# B&R Automation Studio project NAEUL004C00R13L518F00 (part 13)

#### Act_OptP0202InsertRmvMag.st
```iecst
ACTION Act_OptP0202InsertRmvMag:

	//Insert & Removed Magazine Manually Without Button Control
//	IF p_tyNtParamCurr.bProjBtnInsertRmvMag = FALSE THEN
//
//		IF p_bOpsStatusRun AND p_bOpsMagConvUL1InitDone THEN
//
//			fbMag1EntrySenOnTm(IN := p_tyDI.bMagPresentSen1 OR p_tyDI.bMagConvEntSen1);
//
//			IF bNewMag1 = FALSE AND bRlsMag1 = FALSE THEN
//				IF p_bOpsMagConvUL1NewMagAllw AND fbMag1EntrySenOnTm.Q AND NOT p_bOpsMagConvUL1MagExitedWait THEN
//					bNewMag1	:= TRUE;
//				END_IF
//
//				IF p_bOpsMagConvUL1RlsMagAllw AND p_tyDI.bMagPresentSen1 AND p_tyDI.bOutShutterCloseRS AND p_tyBuffer1BffrStat.bBffrFull THEN
//					bRlsMag1	:= TRUE;
//				END_IF
//			END_IF
//
//			IF bNewMag1 = TRUE THEN
//
//				IF p_tyDI.bMag1FixedClampRS = TRUE AND p_tyDI.bMag1RemoteClampRS = TRUE THEN
//					bNewMag1	:= FALSE;
//				END_IF
//
//			ELSIF bRlsMag1 = TRUE THEN
//
//				IF p_tyDI.bMag1FixedUnclampRS = TRUE AND p_tyDI.bMag1RemoteUnclampRS = TRUE AND p_tyDI.bMagConvEntSen1 = TRUE THEN
//					bRlsMag1	:= FALSE;
//				END_IF
//
//			END_IF
//
//		ELSE
//
//			bNewMag1	:= FALSE;
//			bRlsMag1	:= FALSE;
//
//			fbMag1EntrySenOnTm(IN := FALSE);
//
//		END_IF
//
//	END_IF

END_ACTION
```

#### Act_OptP0202RstMnl.st
```iecst
ACTION Act_OptP0202RstMnl:

	IF eCurrPage <> UIP0202OpsMag1 AND eCurrPage <> UIP0003MMenu THEN
		bNewMag1	:= FALSE;
		bRlsMag1	:= FALSE;
		tyP0202OpsMag1.tyOps.tyBtnChgMag.bValue	:= FALSE;
		tyP0202OpsMag1.tyOps.tyBtnChgMag.bRtLk	:= FALSE;
		tyP0202OpsMag1.tyOps.tyBitmapChgMag.usiValueIdx	:= 0;

		tyP0003MMenu.tyMMenuBtn.tyBtnRlsNewMag1.bValue := FALSE;
		tyP0003MMenu.tyMMenuBtn.tyBtnRlsNewMag1.bRtLk  := FALSE;
		tyP0003MMenu.tyMMenuBtn.tyBtnRlsNewMag1.usiBitmapIdx := 0;
	END_IF

END_ACTION
```

#### Act_OptP0202Lane1ChgMag.st
```iecst
ACTION Act_OptP0202Lane1ChgMag:

	tyP0202OpsMag1.tyChgMag.tyBtnChgMag.bRtLk				:= FALSE;

	tChgMag ( IN:= tyP0202OpsMag1.tyChgMag.tyBtnChgMag.bValue = TRUE OR  FALSE , PT:=T#3s0ms);

	IF tChgMag.IN = TRUE THEN

	fbChgMagBlinkTm(IN := TRUE);

		IF fbChgMagBlinkTm.Q THEN
			fbChgMagBlinkTm(IN := FALSE);

			IF (tyP0202OpsMag1.tyChgMag.tyBitmapChgMag.usiValueIdx = 1) THEN
				tyP0202OpsMag1.tyChgMag.tyBitmapChgMag.usiValueIdx		:= 0;
			ELSE
				tyP0202OpsMag1.tyChgMag.tyBitmapChgMag.usiValueIdx		:= 1;
			END_IF
		END_IF
	ELSIF bChgMag = FALSE THEN

		tyP0202OpsMag1.tyChgMag.tyBitmapChgMag.usiValueIdx		:= 0;
	END_IF

	IF tChgMag.Q = TRUE THEN //(tyP0200OpsGen.tyChgMag.tyBtnChgMag.bRtCompl = TRUE) OR (tyP0202OpsMag1.tyChgMag.tyBtnChgMag.bRtCompl = TRUE)
	//	OR (tyP0203OpsMag2.tyChgMag.tyBtnChgMag.bRtCompl = TRUE)	OR (tyP0204OpsOutMagConv.tyChgMag.tyBtnChgMag.bRtCompl = TRUE) THEN

		tyP0202OpsMag1.tyChgMag.tyBitmapChgMag.usiValueIdx	:= 1;

		tyP0202OpsMag1.tyChgMag.tyBtnChgMag.bRtCompl			:= FALSE;

		bChgMag			:= TRUE;

//	ELSIF EDGEPOS(p_bFollower2SetBffrFull) THEN
//		bFllw2SetFull	:= TRUE;
//	ELSIF EDGEPOS(p_tyDI.bChgMagSig) THEN
//		bChgMagSig		:= TRUE;
	END_IF

	IF (p_bOpsOutMagConvStepInitDone AND p_bOpsStatusRun = TRUE) AND bChgMag = TRUE THEN

		eBuffer1Act			:= BufferActSetFull;

		IF p_eBuffer1Stat = BufferActSetFull AND p_eBuffer1Status = Done THEN
			eBuffer1Act		:= BufferActIdle;

			bChgMag			:= FALSE;

		END_IF

//	ELSIF bFllw2SetFull = TRUE THEN
//		eBufferAct			:= BufferActSetFull;
//
//		IF p_eBufferStat = BufferActSetFull AND p_eBufferStatus = Done THEN
//			eBufferAct		:= BufferActIdle;
//
//			bFllw2SetFull	:= FALSE;
//		END_IF

	ELSIF (p_bOpsOutMagConvStepInitDone AND p_bOpsStatusRun = TRUE) AND bChgMagSig THEN //ADAM Feature

		eBuffer1Act			:= BufferActSetFull;

		IF p_eBuffer1Stat = BufferActSetFull AND p_eBuffer1Status = Done THEN
			eBuffer1Act		:= BufferActIdle;

			bChgMagSig		:= FALSE;

		END_IF

	END_IF

	IF p_tyDI.bLifterLmtSW = TRUE THEN
		fUIInRtStatHide(ADR(tyP0202OpsMag1.tyChgMag.tyBtnChgMag.uiMaskRtStat));
	ELSE
		fUIInRtStatOff(ADR(tyP0202OpsMag1.tyChgMag.tyBtnChgMag.uiMaskRtStat));
	END_IF

	//Manual unload magazine-------------------------------------------------------------------------------------------------------------
	IF p_bOpsRun THEN
		IF tyP0202OpsMag1.tyChgMag.tyBtnMnlUnloadMag.bValue THEN
			bOpsMnlUnloadMag := TRUE;
		ELSE
			bOpsMnlUnloadMag := FALSE;
		END_IF
	ELSE
		tyP0202OpsMag1.tyChgMag.tyBtnMnlUnloadMag.bValue := FALSE;
		bOpsMnlUnloadMag := FALSE;
	END_IF

	IF p_bOpsRun AND p_eOutMagConvStatus <> Busy THEN
		fUIInRtStatHide (ADR(tyP0202OpsMag1.tyChgMag.tyBtnMnlUnloadMag.uiMaskRtStat));
	ELSE
		fUIInRtStatOff (ADR(tyP0202OpsMag1.tyChgMag.tyBtnMnlUnloadMag.uiMaskRtStat));
	END_IF

END_ACTION
```

#### Act_OptP0202AIVDat.st - not listed in the package file held
```iecst
ACTION Act_OptP0202AIVDat:

	//Show Change Mag Button only in Manual Exchane Mode
	// insert and remove temporaray replace change magazine button
	tyP0202OpsMag1.tyOps.tyBtnChgMag.uiRtStat.0 := (p_tyMcParamCurr.eMagExMode = McSetMagXcAutoMode AND p_tyMcParamCurr.eAGVComProtocol <> McSetAGVCommDisabled OR p_tyNtParamCurr.bProjLifterMagPlatform) (*OR (p_tyNtParamCurr.bProjBtnInsertRmvMag = FALSE)*);
	tyP0202OpsMag1.tyOps.tyBitmapChgMag.uiRtStat.0 := p_tyMcParamCurr.eMagExMode = McSetMagXcAutoMode  AND p_tyMcParamCurr.eAGVComProtocol <> McSetAGVCommDisabled OR p_tyNtParamCurr.bProjLifterMagPlatform (*OR (p_tyNtParamCurr.bProjBtnInsertRmvMag = FALSE)*);

	//LED Wifi
	tyP0202OpsMag1.tyOps.tyBtnAIVWifi.bValue	:= p_bAGVOnline;

	//Change Magazine
	IF p_tyNtParamCurr.bProjBtnInsertRmvMag = TRUE THEN

		IF EDGENEG(p_bOpsStatusRun) THEN
			bNewMag1	:= FALSE;
			tyP0202OpsMag1.tyOps.tyBtnChgMag.bRtLk	:= FALSE;
			tyP0202OpsMag1.tyOps.tyBtnChgMag.bRtCompl	:= FALSE;
			tyP0202OpsMag1.tyOps.tyBtnChgMag.bValue		:= FALSE;
		END_IF

		IF tyP0202OpsMag1.tyOps.tyBtnChgMag.bRtCompl = TRUE THEN
			tyP0202OpsMag1.tyOps.tyBtnChgMag.bRtCompl	:= FALSE;
			bNewMag1	:= p_bOpsMagConvUL1NewMagAllw;
			bRlsMag1	:= p_bOpsMagConvUL1RlsMagAllw;
		END_IF

		IF bNewMag1 = TRUE THEN
			tyP0202OpsMag1.tyOps.tyBitmapChgMag.usiValueIdx	:= 1;
			IF p_tyDI.bMag1FixedUnclampRS = FALSE THEN
				bNewMag1	:= FALSE;
				tyP0202OpsMag1.tyOps.tyBtnChgMag.bValue	:= FALSE;
				tyP0202OpsMag1.tyOps.tyBtnChgMag.bRtLk	:= FALSE;
				tyP0202OpsMag1.tyOps.tyBitmapChgMag.usiValueIdx	:= 0;
			END_IF

		ELSIF bRlsMag1 = TRUE THEN
			tyP0202OpsMag1.tyOps.tyBitmapChgMag.usiValueIdx	:= 1;
			IF p_tyNtParamCurr.eCustomerReq = Siemens THEN
				IF p_bOpsMagConvUL1EjectMESStep THEN //(p_bOpsMagConvUL1EjectMESStep AND p_bOpsMagConvUL1EjectMagNotAllw)
					//OR THEN //FOR MES
					bRlsMag1	:= FALSE;
					tyP0202OpsMag1.tyOps.tyBtnChgMag.bValue	:= FALSE;
					tyP0202OpsMag1.tyOps.tyBtnChgMag.bRtLk	:= FALSE;
					tyP0202OpsMag1.tyOps.tyBitmapChgMag.usiValueIdx	:= 0;
				END_IF
			ELSIF p_tyDI.bMag1FixedUnclampRS = TRUE AND p_tyDI.bMagPresentSen1 = FALSE  THEN //for Siemen testing
				bRlsMag1	:= FALSE;
				tyP0202OpsMag1.tyOps.tyBtnChgMag.bValue	:= FALSE;
				tyP0202OpsMag1.tyOps.tyBtnChgMag.bRtLk	:= FALSE;
				tyP0202OpsMag1.tyOps.tyBitmapChgMag.usiValueIdx	:= 0;
			END_IF

		ELSIF p_bAlarmErr THEN
			bNewMag1	:= FALSE;
			bRlsMag1	:= FALSE;
			tyP0202OpsMag1.tyOps.tyBtnChgMag.bValue	:= FALSE;
			tyP0202OpsMag1.tyOps.tyBtnChgMag.bRtLk	:= FALSE;
			tyP0202OpsMag1.tyOps.tyBitmapChgMag.usiValueIdx	:= 0;
		END_IF

		IF p_tyDI.bMagPresentSen1 AND p_tyDI.bMagConvEntSen1 = FALSE THEN
			tyP0202OpsMag1.tyOps.tyBtnChgMag.usiTxtIdx	:= 1;
		ELSE
			tyP0202OpsMag1.tyOps.tyBtnChgMag.usiTxtIdx	:= 0;
		END_IF

		IF (p_bOpsMagConvUL1NewMagAllw AND p_tyBuffer1BffrStat.bBffrMty)
			OR p_bOpsMagConvUL1RlsMagAllw
			OR p_bBufferMagRemoved1
			THEN //AND p_tyDI.bOutShutterCloseRS
			fUIInRtStatHide(ADR(tyP0202OpsMag1.tyOps.tyBtnChgMag.uiMaskRtStat));
		ELSE
			fUIInRtStatOff(ADR(tyP0202OpsMag1.tyOps.tyBtnChgMag.uiMaskRtStat));
		END_IF

	END_IF

END_ACTION
```

#### Act_EntP0203Disp.st
```iecst
ACTION Act_EntP0203Disp:
	//Access Address
	p_tyC0004Navi ACCESS ADR(tyP0203OpsMag2.tyNaviBack);

	p_tyC0005Main ACCESS ADR(tyCommon.tyMain);

	p_tyC0007Notif ACCESS ADR(tyCommon.tyNotif);

	p_tyC0008MsgBox ACCESS ADR(tyP0203OpsMag2.tyMsgBoxHide);

	p_tyC0009Info ACCESS ADR(tyCommon.tyInfo);

	p_tyC0011RcpPopUp ACCESS ADR(tyP0203OpsMag2.tyRcpPopUp);

	p_tyP0203Ops ACCESS ADR(tyP0203OpsMag2.tyOps);
	p_tyP0203IOMonitor ACCESS ADR(tyP0203OpsMag2.tyIOMonitor);
	p_tyP0203BypsInitConv ACCESS ADR(tyP0203OpsMag2.tyBypsInitConv);
	p_tyP0203Param ACCESS ADR(tyP0203OpsMag2.tyParam);
	p_tyP0203ChgMagL2 ACCESS ADR(tyP0203OpsMag2.tyChgMag);

	//Display
	fUIInRtStatHide(ADR(tyP0203OpsMag2.tyIOMonitor.tyLyr.uiRtStat));
	fUIInRtStatHide(ADR(tyP0203OpsMag2.tyParam.tyLyr.uiRtStat));

	tyP0203OpsMag2.tyOps.tyBtnChgParam.uiRtStat.0	:= NOT(p_tyMcParamCurr.bChgParamEn);

	IF p_tyNtParamCurr.bMagAutoVerifyPrep = FALSE THEN
		tyP0203OpsMag2.tyIOMonitor.tyBtnMag2FixedClmpRS.usiTxtIdx	:= 68;
		tyP0203OpsMag2.tyIOMonitor.tyBtnMag2FixedUnclmpRS.usiTxtIdx:= 68;
		tyP0203OpsMag2.tyIOMonitor.tyBtnMag2RmtClmpRS.usiTxtIdx	:= 0;
		tyP0203OpsMag2.tyIOMonitor.tyBtnMag2RmtUnclmpRS.usiTxtIdx:= 0;
		tyP0203OpsMag2.tyIOMonitor.tyBtnMag2FixedClampCtrl.usiTxtIdx:= 34;
		tyP0203OpsMag2.tyIOMonitor.tyBtnMag2RemoteClampCtrl.usiTxtIdx:= 18;
	ELSE
		//	tyP0203OpsMag2.tyIOMonitor.tyBtnMag2FixedClmpRS.usiTxtIdx	:= 74;
		tyP0203OpsMag2.tyIOMonitor.tyBtnMag2FixedUnclmpRS.usiTxtIdx:= 68;
		//	tyP0203OpsMag2.tyIOMonitor.tyBtnMag2RmtClmpRS.usiTxtIdx	:= 51;
		//	tyP0203OpsMag2.tyIOMonitor.tyBtnMag2RmtUnclmpRS.usiTxtIdx:= 50;
		tyP0203OpsMag2.tyIOMonitor.tyBtnMag2FixedClampCtrl.usiTxtIdx:= 34;
			tyP0203OpsMag2.tyIOMonitor.tyBtnMag2RemoteClampCtrl.usiTxtIdx:= 18;

	END_IF

	tyP0203OpsMag2.tyParam.tyNumMaxSlt.diValueMax	:= p_tyMagRcpCurrRcp.diTtlSlt;

END_ACTION
```

#### Act_OptP0203Navi.st
```iecst
ACTION Act_OptP0203Navi:

	IF tyP0203OpsMag2.tyNaviBack.tyBtnBack.bRtCompl = TRUE THEN
		tyP0203OpsMag2.tyNaviBack.tyBtnBack.bRtCompl	:= FALSE;
		tyP0203OpsMag2.tyNaviBack.tyBtnBack.bValue		:= FALSE;

		eChgPage	:= UIP0200OpsGen;

	END_IF

END_ACTION
```

#### Act_OptP0203ChgPage.st
```iecst
ACTION Act_OptP0203ChgPage:

	IF tyP0203OpsMag2.tyOps.tyHotspotMagInfo.bRtCompl = TRUE THEN
		tyP0203OpsMag2.tyOps.tyHotspotMagInfo.bRtCompl	:= FALSE;

		eChgPage	:= UIP0800MagInfo;
	END_IF

END_ACTION
```

#### Act_OptP0203UpdtDat.st
```iecst
ACTION Act_OptP0203UpdtDat:

	//Status
	fbMcStatUpdtTm(IN := TRUE);
	IF fbMcStatUpdtTm.Q = TRUE THEN
		fbMcStatUpdtTm(IN := FALSE);

//		IF p_tyNtParamCurr.bProjMag2ConvPrep = FALSE THEN
//			tyP0203OpsMag2.tyOps.tyStringMcStat.sValue	:= p_sOpsMagUL2StepTxt;
//		ELSE
//			tyP0203OpsMag2.tyOps.tyStringMcStat.sValue	:= p_sOpsMagConvUL2StepTxt;
//		END_IF

		IF p_tyNtParamCurr.bProjLifterMagPlatform AND p_tyNtParamCurr.bProjMagConvLane2Prep THEN
			IF p_bOpsLifMagULStepIdle2 THEN
				tyP0203OpsMag2.tyOps.tyStringMcStat.sValue		:= p_sOpsLifMagULStepTxt; //main text
			ELSE
				tyP0203OpsMag2.tyOps.tyStringMcStat.sValue		:= p_sOpsLifMagULStepTxt1; //Lifter 2 text
			END_IF
		ELSIF p_tyNtParamCurr.bProjLifterMagPlatform THEN
			tyP0203OpsMag2.tyOps.tyStringMcStat.sValue		:= p_sOpsLifMagULStepTxt;
		ELSE
			tyP0203OpsMag2.tyOps.tyStringMcStat.sValue	:= p_sOpsMagConvUL2StepTxt;
		END_IF

	END_IF

	//Width
	IF p_tyNtParamCurr.bAWPrep = TRUE AND p_tyMcParamCurr.bAWDis = FALSE THEN
		tyP0203OpsMag2.tyOps.tyNumWidth.diValue		:= p_tyMcParamCurr.diWidthAtHmPosInUM - p_diAWOpenActualPos;
		tyP0203OpsMag2.tyOps.tyNumWidth2.diValue	:= p_tyMcParamCurr.diWidthAtHmPosInUM - p_diAWOpenActualPos;
	ELSE
		tyP0203OpsMag2.tyOps.tyNumWidth.diValue		:= p_tyProdRcpCurrRcp1.diWidthInUM;
		tyP0203OpsMag2.tyOps.tyNumWidth2.diValue		:= p_tyProdRcpCurrRcp1.diWidthInUM2;
	END_IF

	//Program Info

	IF p_bMcParamAutoRcpDisable OR p_bNtParamAutoRcpF1ArbitraryType THEN
		tyP0203OpsMag2.tyOps.tyTxtMod.usiValueIdx	:= p_tyProdRcpCurrRcp2.usiMcMod;
		tyP0203OpsMag2.tyOps.tyNumMinSltRange.diValue	:= p_tyProdRcpCurrRcp2.diMinSltValue;
		tyP0203OpsMag2.tyOps.tyNumMaxSltRange.diValue	:= p_tyProdRcpCurrRcp2.diMaxSltValue;
		tyP0203OpsMag2.tyOps.tyBtnToptoBtm.bValue		:= p_tyProdRcpCurrRcp2.bTopToBtm;
		tyP0203OpsMag2.tyOps.tyNumPitch.diValue			:= p_tyProdRcpCurrRcp2.diPitch;
		tyP0203OpsMag2.tyOps.tyStringProdNm.sValue		:= p_tyProdRcpCurrRcp2.sRcpNm;
	ELSE  //FALSE AutoRcp Mode
		tyP0203OpsMag2.tyOps.tyTxtMod.usiValueIdx	:= p_tyProdRcpCurrRcp0.usiMcMod;
		tyP0203OpsMag2.tyOps.tyNumMinSltRange.diValue	:= pa_tyMagProps[2].diMinSlt;
		tyP0203OpsMag2.tyOps.tyNumMaxSltRange.diValue	:= pa_tyMagProps[2].diMaxSlt;
		tyP0203OpsMag2.tyOps.tyBtnToptoBtm.bValue		:= p_tyProdRcpCurrRcp0.bTopToBtm;
		tyP0203OpsMag2.tyOps.tyNumPitch.diValue			:= pa_tyMagProps[2].diPitch;
		IF p_tyNtParamCurr.eAutoRcpPrecededBy =  PrecededBySelf THEN
			tyP0203OpsMag2.tyOps.tyStringProdNm.sValue		:= pa_tyAutoRcpBrdProps[2].sProductTypeId;
		ELSIF p_tyNtParamCurr.eAutoRcpPrecededBy =  PrecededByF1 THEN
			tyP0203OpsMag2.tyOps.tyStringProdNm.sValue		:= pa_tyMagProps[2].sRcpNm;
		END_IF
	END_IF

	//Magazine Info
	tyP0203OpsMag2.tyOps.tyStringMagNm.sValue	:= p_tyMagRcpCurrRcp.sRcpNm;

	IF p_bBuffer2MagPresent = TRUE THEN
		IF p_tyNtParamCurr.eCustomerReq = Siemens AND p_iOpsMagConvUL2MESAcptCond <= 0 AND  p_tyMcParamCurr.bMESEn THEN
			tyP0203OpsMag2.tyOps.tyNumMag2AvlQty.diValue	:= 0;
			tyP0203OpsMag2.tyOps.tyNumMag2TtlSlt.diValue	:= 0;
		ELSE
			tyP0203OpsMag2.tyOps.tyNumMag2AvlQty.diValue	:= p_tyBuffer2BffrStat.diTtlBrdCap - (p_tyBuffer2BffrStat.diTtlGdBrd + p_tyBuffer2BffrStat.diTtlBadBrd);
			tyP0203OpsMag2.tyOps.tyNumMag2TtlSlt.diValue	:= p_tyBuffer2BffrStat.diTtlBrdCap;
		END_IF
	ELSE
		tyP0203OpsMag2.tyOps.tyNumMag2AvlQty.diValue	:= 0;
		tyP0203OpsMag2.tyOps.tyNumMag2TtlSlt.diValue	:= 0;
	END_IF

	//Magazine Present States
	IF p_bBuffer2MagPresent = TRUE THEN

		IF p_tyBuffer2BffrStat.bBffrFull = TRUE THEN
			tyP0203OpsMag2.tyOps.tyTxtMag2Stat.usiValueIdx := 2;
			tyP0203OpsMag2.tyOps.tyTxtMag2Stat.usiColor	   := 1;
		ELSIF p_tyBuffer2BffrStat.bBffrMty = TRUE THEN
			tyP0203OpsMag2.tyOps.tyTxtMag2Stat.usiValueIdx := 1;
			tyP0203OpsMag2.tyOps.tyTxtMag2Stat.usiColor	   := 0;
		ELSE
			tyP0203OpsMag2.tyOps.tyTxtMag2Stat.usiValueIdx := 3;
			tyP0203OpsMag2.tyOps.tyTxtMag2Stat.usiColor	   := 0;
		END_IF

	ELSE
		tyP0203OpsMag2.tyOps.tyTxtMag2Stat.usiValueIdx := 0;
		tyP0203OpsMag2.tyOps.tyTxtMag2Stat.usiColor	   := 1;
	END_IF

	//Product Recipe 254
	tyP0203OpsMag2.tyOps.tyHotspotShowLRcp.uiRtStat.0 := NOT(tyP0203OpsMag2.tyOps.tyStringProdNm.sValue <> '');

	IF tyP0203OpsMag2.tyOps.tyHotspotShowLRcp.bRtCompl = TRUE THEN
		tyP0203OpsMag2.tyOps.tyHotspotShowLRcp.bRtCompl := FALSE;

		fUIInRtStatOff(ADR(tyP0203OpsMag2.tyRcpPopUp.tyLyr.uiRtStat));

		tyP0203OpsMag2.tyRcpPopUp.tyStringInfo.sValue  := p_tyProdRcpCurrRcp1.sRcpNm;

	ELSIF tyP0203OpsMag2.tyRcpPopUp.tyHotspotClose.bRtCompl = TRUE THEN
		tyP0203OpsMag2.tyRcpPopUp.tyHotspotClose.bRtCompl := FALSE;

		fUIInRtStatHide(ADR(tyP0203OpsMag2.tyRcpPopUp.tyLyr.uiRtStat));

	END_IF

END_ACTION
```

#### Act_OptP0203IOMonitor.st
```iecst
ACTION Act_OptP0203IOMonitor:

	IF tyP0203OpsMag2.tyOps.tyHotspotIOMonitor.bRtCompl = TRUE THEN
		tyP0203OpsMag2.tyOps.tyHotspotIOMonitor.bRtCompl	:= FALSE;

		fUIInRtStatOff(ADR(tyP0203OpsMag2.tyIOMonitor.tyLyr.uiRtStat));

		p_tyC0004Navi ACCESS ADR(tyP0203OpsMag2.tyNaviHide);

	ELSIF tyP0203OpsMag2.tyIOMonitor.tyHotspotClose.bRtCompl = TRUE THEN
		tyP0203OpsMag2.tyIOMonitor.tyHotspotClose.bRtCompl	:= FALSE;

		fUIInRtStatHide(ADR(tyP0203OpsMag2.tyIOMonitor.tyLyr.uiRtStat));

		p_tyC0004Navi ACCESS ADR(tyP0203OpsMag2.tyNaviBack);

	END_IF

	IF tyP0203OpsMag2.tyIOMonitor.tyLyr.uiRtStat.0 = FALSE THEN

		//Digital Input
		tyP0203OpsMag2.tyIOMonitor.tyBtnSafetyRlySig.bValue				:= p_tyDI.bSafetyRlySig;
		tyP0203OpsMag2.tyIOMonitor.tyBtnEStop.bValue					:= p_tyDI.bEStopSig;
		tyP0203OpsMag2.tyIOMonitor.tyBtnCoverSWSig.bValue				:= p_tyDI.bCoverSWSig;
		tyP0203OpsMag2.tyIOMonitor.tyBtnUBAA.bValue						:= p_tyDI.bUBAA;
		tyP0203OpsMag2.tyIOMonitor.tyBtnUBAB.bValue						:= p_tyDI.bUBAB;
		tyP0203OpsMag2.tyIOMonitor.tyBtnUBAAStat.bValue					:= p_tyDI.bUBAAStat;
		tyP0203OpsMag2.tyIOMonitor.tyBtnUBABStat.bValue					:= p_tyDI.bUBABStat;
		tyP0203OpsMag2.tyIOMonitor.tyBtnOvenInfeedSigA.bValue			:= p_tyDI.bOvenInfeedSigA;
		tyP0203OpsMag2.tyIOMonitor.tyBtnOvenInfeedSigB.bValue			:= p_tyDI.bOvenInfeedSigB;
		tyP0203OpsMag2.tyIOMonitor.tyBtnMag2FixedClmpRS.bValue			:= p_tyDI.bMag2FixedClampRS;
		tyP0203OpsMag2.tyIOMonitor.tyBtnMag2FixedUnclmpRS.bValue		:= p_tyDI.bMag2FixedUnclampRS;
		tyP0203OpsMag2.tyIOMonitor.tyBtnMag2RmtClmpRS.bValue			:= p_tyDI.bMag2RemoteClampRS;
		tyP0203OpsMag2.tyIOMonitor.tyBtnMag2RmtUnclmpRS.bValue			:= p_tyDI.bMag2RemoteUnclampRS;
		tyP0203OpsMag2.tyIOMonitor.tyBtnMag2ConvEntrySen.bValue			:= p_tyDI.bMagConvEntSen2;
		tyP0203OpsMag2.tyIOMonitor.tyBtnMag2PresentSen.bValue			:= p_tyDI.bMagPresentSen2;
		tyP0203OpsMag2.tyIOMonitor.tyBtnMag2AIVInPosSen1.bValue			:= p_tyDI.bMag2AIVInPosSen1;
		tyP0203OpsMag2.tyIOMonitor.tyBtnMag2AIVInPosSen2.bValue			:= p_tyDI.bMag2AIVInPosSen2;
		tyP0203OpsMag2.tyIOMonitor.tyBtnMag2OrientationChkSen1.bValue	:= p_tyDI.bMag2OrientChkSen1;
		tyP0203OpsMag2.tyIOMonitor.tyBtnMag2OrientationChkSen2.bValue	:= p_tyDI.bMag2OrientChkSen2;

		tyP0203OpsMag2.tyIOMonitor.tyBtnSelUnclampRS.bValue				:= p_tyDI.bMag2SelUnClampRS;

		tyP0203OpsMag2.tyIOMonitor.tyBtnCAB717Sen.bValue				:= p_tyDI.bMagConvCAB717MagSen2;
//		tyP0203OpsMag2.tyIOMonitor.tyBtnHeightSen.bValue				:= p_tyDI.bMagConvHeightSen2;
		tyP0203OpsMag2.tyIOMonitor.tyBtnMagSmallSen.bValue				:= p_tyDI.bMagConvSmallMagSen2;
		tyP0203OpsMag2.tyIOMonitor.tyBtnMagLargeSen.bValue				:= p_tyDI.bMagConvLargeMagSen2;
		tyP0203OpsMag2.tyIOMonitor.tyBtnCurtainSen.bValue				:= p_tyDI.bCurtainSen;
		tyP0203OpsMag2.tyIOMonitor.tyBtnCurtainSenPB.bValue				:= p_tyDI.bCurtainSenPB;
		tyP0203OpsMag2.tyIOMonitor.tyBtnMag2DetSen.bValue				:= p_tyDI.bMag2FixedClampSen;

		IF p_tyNtParamCurr.bMagAutoVerifyPrep = TRUE THEN
			tyP0203OpsMag2.tyIOMonitor.tyBtnHeightSen.bValue			:= p_tyDI.bMagConvHeightSen2;
		ELSE
			tyP0203OpsMag2.tyIOMonitor.tyBtnHeightSen.bValue			:= p_tyDI.bHighMagDetSen2;
		END_IF

		//Digital Output
		tyP0203OpsMag2.tyIOMonitor.tyBtnSafetyRlyRst.bValue				:= p_tyDO.bSafetyRlyRst;
		tyP0203OpsMag2.tyIOMonitor.tyBtnTLGreen.bValue					:= p_tyDO.bTLGreen;
		tyP0203OpsMag2.tyIOMonitor.tyBtnTLAmber.bValue					:= p_tyDO.bTLAmber;
		tyP0203OpsMag2.tyIOMonitor.tyBtnTLRed.bValue					:= p_tyDO.bTLRed;
		tyP0203OpsMag2.tyIOMonitor.tyBtnBuzzer.bValue					:= p_tyDO.bBuzzer;
		tyP0203OpsMag2.tyIOMonitor.tyBtnUSBA.bValue						:= p_tyDO.bUSBA;
		tyP0203OpsMag2.tyIOMonitor.tyBtnUSBB.bValue						:= p_tyDO.bUSBB;
		tyP0203OpsMag2.tyIOMonitor.tyBtnOvenInfoSigA.bValue				:= p_tyDO.bOvenInfoSigA;
		tyP0203OpsMag2.tyIOMonitor.tyBtnOvenInfoSigB.bValue				:= p_tyDO.bOvenInfoSigB;
		tyP0203OpsMag2.tyIOMonitor.tyBtnMag2FixedClampCtrl.bValue		:= p_tyDO.bMag2FixedClampCtrl;
		tyP0203OpsMag2.tyIOMonitor.tyBtnMag2RemoteClampCtrl.bValue		:= p_tyDO.bMag2RemoteClampCtrl;
		tyP0203OpsMag2.tyIOMonitor.tyBtnMag2ConvMtrIn.bValue			:= p_tyDO.bMag2ConvMtrIn;
		tyP0203OpsMag2.tyIOMonitor.tyBtnMag2ConvMtrOut.bValue			:= p_tyDO.bMag2ConvMtrOut;
		tyP0203OpsMag2.tyIOMonitor.tyBtnMagSelClampCtrl.bValue			:= p_tyDO.bMag2SelClampCtrl;
		//tyP0203OpsMag2.tyIOMonitor.tyBtnMagSelUnClampCtrl.bValue		:= p_tyDO.bMag2SelUnClampCtrl;
		tyP0203OpsMag2.tyIOMonitor.tyBtnCurtainSenPBLED.bValue			:= p_tyDO.bBypCurtainPBLED;
	END_IF

END_ACTION
```

#### Act_OptP0203_P0003AIVDat.st
```iecst
ACTION Act_OptP0203_P0003AIVDat:

	//Show Change Mag Button only in Manual Exchane Mode
	tyP0203OpsMag2.tyOps.tyBtnChgMag.uiRtStat.0 := p_tyMcParamCurr.eMagExMode = McSetMagXcAutoMode  AND p_tyMcParamCurr.eAGVComProtocol <> McSetAGVCommDisabled OR p_tyNtParamCurr.bProjLifterMagPlatform;
	tyP0203OpsMag2.tyOps.tyBitmapChgMag.uiRtStat.0 := p_tyMcParamCurr.eMagExMode = McSetMagXcAutoMode  AND p_tyMcParamCurr.eAGVComProtocol <> McSetAGVCommDisabled OR p_tyNtParamCurr.bProjLifterMagPlatform;

	//LED Wifi
	tyP0203OpsMag2.tyOps.tyBtnAIVWifi.bValue	:= p_bAGVOnline;

	//Change Magazine
	IF p_tyNtParamCurr.bProjBtnInsertRmvMag = TRUE THEN

		IF EDGENEG(p_bOpsStatusRun) THEN
			bNewMag2	:= FALSE;
			tyP0203OpsMag2.tyOps.tyBtnChgMag.bRtLk	:= FALSE;
			tyP0203OpsMag2.tyOps.tyBtnChgMag.bRtCompl	:= FALSE;
			tyP0003MMenu.tyMMenuBtn.tyBtnRlsNewMag2.bRtLk    := FALSE;
			tyP0003MMenu.tyMMenuBtn.tyBtnRlsNewMag2.bRtCompl := FALSE;
			tyP0203OpsMag2.tyOps.tyBtnChgMag.bValue		:= FALSE;
			tyP0003MMenu.tyMMenuBtn.tyBtnRlsNewMag2.bValue	:= FALSE;
		END_IF

		IF tyP0203OpsMag2.tyOps.tyBtnChgMag.bRtCompl = TRUE OR tyP0003MMenu.tyMMenuBtn.tyBtnRlsNewMag2.bRtCompl THEN
			tyP0203OpsMag2.tyOps.tyBtnChgMag.bRtCompl	:= FALSE;
			tyP0003MMenu.tyMMenuBtn.tyBtnRlsNewMag2.bRtCompl := FALSE;
			bNewMag2	:= p_bOpsMagConvUL2NewMagAllw;
			bRlsMag2	:= p_bOpsMagConvUL2RlsMagAllw;
		END_IF

		IF bNewMag2 = TRUE THEN
			tyP0203OpsMag2.tyOps.tyBitmapChgMag.usiValueIdx	:= 1;
			tyP0003MMenu.tyMMenuBtn.tyBtnRlsNewMag2.usiBitmapIdx := 1;
			IF p_tyDI.bMag2FixedUnclampRS = FALSE THEN
				bNewMag2	:= FALSE;
				tyP0203OpsMag2.tyOps.tyBtnChgMag.bValue	:= FALSE;
				tyP0003MMenu.tyMMenuBtn.tyBtnRlsNewMag2.bValue := FALSE;
				tyP0203OpsMag2.tyOps.tyBtnChgMag.bRtLk	:= FALSE;
				tyP0003MMenu.tyMMenuBtn.tyBtnRlsNewMag2.bRtLk:= FALSE;
				tyP0203OpsMag2.tyOps.tyBitmapChgMag.usiValueIdx	:= 0;
				tyP0003MMenu.tyMMenuBtn.tyBtnRlsNewMag2.usiBitmapIdx := 0;
			END_IF

		ELSIF bRlsMag2 = TRUE THEN
			tyP0203OpsMag2.tyOps.tyBitmapChgMag.usiValueIdx	:= 1;
			tyP0003MMenu.tyMMenuBtn.tyBtnRlsNewMag2.usiBitmapIdx := 1;
			IF p_tyNtParamCurr.eCustomerReq = Siemens  THEN
				IF p_bOpsMagConvUL2EjectMESStep  THEN //FOR MES
					bRlsMag2	:= FALSE;
					tyP0203OpsMag2.tyOps.tyBtnChgMag.bValue	:= FALSE;
					tyP0003MMenu.tyMMenuBtn.tyBtnRlsNewMag2.bValue := FALSE;
					tyP0203OpsMag2.tyOps.tyBtnChgMag.bRtLk	:= FALSE;
					tyP0003MMenu.tyMMenuBtn.tyBtnRlsNewMag2.bRtLk := FALSE;
					tyP0203OpsMag2.tyOps.tyBitmapChgMag.usiValueIdx	:= 0;
					tyP0003MMenu.tyMMenuBtn.tyBtnRlsNewMag2.usiBitmapIdx := 0;
				END_IF
			ELSIF p_tyDI.bMag2FixedUnclampRS = TRUE AND p_tyDI.bMagPresentSen2 = FALSE THEN
				bRlsMag2	:= FALSE;
				tyP0203OpsMag2.tyOps.tyBtnChgMag.bValue	:= FALSE;
				tyP0003MMenu.tyMMenuBtn.tyBtnRlsNewMag2.bValue := FALSE;
				tyP0203OpsMag2.tyOps.tyBtnChgMag.bRtLk	:= FALSE;
				tyP0003MMenu.tyMMenuBtn.tyBtnRlsNewMag2.bRtLk := FALSE;
				tyP0203OpsMag2.tyOps.tyBitmapChgMag.usiValueIdx	:= 0;
				tyP0003MMenu.tyMMenuBtn.tyBtnRlsNewMag2.usiBitmapIdx := 0;
			END_IF

		ELSIF p_bAlarmErr THEN
			bNewMag2	:= FALSE;
			bRlsMag2	:= FALSE;
			tyP0203OpsMag2.tyOps.tyBtnChgMag.bValue	:= FALSE;
			tyP0003MMenu.tyMMenuBtn.tyBtnRlsNewMag2.bValue := FALSE;
			tyP0203OpsMag2.tyOps.tyBtnChgMag.bRtLk	:= FALSE;
			tyP0003MMenu.tyMMenuBtn.tyBtnRlsNewMag2.bRtLk:= FALSE;
			tyP0203OpsMag2.tyOps.tyBitmapChgMag.usiValueIdx	:= 0;
			tyP0003MMenu.tyMMenuBtn.tyBtnRlsNewMag2.usiBitmapIdx := 0;
		END_IF

		IF p_tyDI.bMagPresentSen2 AND p_tyDI.bMagConvEntSen2 = FALSE THEN
			tyP0203OpsMag2.tyOps.tyBtnChgMag.usiTxtIdx	:= 1;
			tyP0003MMenu.tyMMenuBtn.tyBtnRlsNewMag2.usiTxtIdx := 32;
		ELSE
			tyP0203OpsMag2.tyOps.tyBtnChgMag.usiTxtIdx	:= 0;
			tyP0003MMenu.tyMMenuBtn.tyBtnRlsNewMag2.usiTxtIdx := 7;
		END_IF

		IF (p_bOpsMagConvUL2NewMagAllw AND p_tyBuffer2BffrStat.bBffrMty)
			OR p_bOpsMagConvUL2RlsMagAllw
			OR p_bBufferMagRemoved2
			THEN //AND p_tyDI.bOutShutterCloseRS
			fUIInRtStatHide(ADR(tyP0203OpsMag2.tyOps.tyBtnChgMag.uiMaskRtStat));
			fUIInRtStatHide(ADR(tyP0003MMenu.tyMMenuBtn.tyBtnRlsNewMag2.uiMaskRtStat));
		ELSE
			fUIInRtStatOff(ADR(tyP0203OpsMag2.tyOps.tyBtnChgMag.uiMaskRtStat));
			fUIInRtStatOff(ADR(tyP0003MMenu.tyMMenuBtn.tyBtnRlsNewMag2.uiMaskRtStat));
		END_IF

	END_IF

END_ACTION
```

#### Act_OptP0203ChgParam.st
```iecst
ACTION Act_OptP0203ChgParam:

	tyP0203OpsMag2.tyParam.tyNumMinSlt.diValueMax		:= tyP0203OpsMag2.tyParam.tyNumMaxSlt.diValue;
	tyP0203OpsMag2.tyParam.tyNumMaxSlt.diValueMin		:= tyP0203OpsMag2.tyParam.tyNumMinSlt.diValue;
	tyP0203OpsMag2.tyParam.tyNumPitch.diValueMax		:= tyP0203OpsMag2.tyParam.tyNumMaxSlt.diValue - tyP0203OpsMag2.tyParam.tyNumMinSlt.diValue + 1;
	tyP0203OpsMag2.tyParam.tyNumPitch.diValueMin		:= 1;
	tyP0203OpsMag2.tyOps.tyBtnChgParam.uiRtStat.0	:= NOT(p_tyMcParamCurr.bChgParamEn);

	tyP0203OpsMag2.tyParam.tyNumPshrExtSpeed.diValueMin 	:= p_tyNtParamCurr.tyProdRcpMtrPshrExtSpd.diMin;
	tyP0203OpsMag2.tyParam.tyNumPshrExtSpeed.diValueMax 	:= p_tyNtParamCurr.tyProdRcpMtrPshrExtSpd.diMax;
	tyP0203OpsMag2.tyParam.tyNumPshrExtTorque.diValueMin	:= p_tyNtParamCurr.tyProdRcpMtrPshrExtTorq.diMin;
	tyP0203OpsMag2.tyParam.tyNumPshrExtTorque.diValueMax	:= p_tyNtParamCurr.tyProdRcpMtrPshrExtTorq.diMax;
	tyP0203OpsMag2.tyParam.tyNumPshrExtSpeed.uiRtStat.0		:= NOT p_tyNtParamCurr.bProjMotorizedPusherPrep;
	tyP0203OpsMag2.tyParam.tyNumPshrExtTorque.uiRtStat.0	:= NOT p_tyNtParamCurr.bProjMotorizedPusherPrep;

	IF (tyP0203OpsMag2.tyOps.tyNumWidth.diValue) <> 0 THEN
		tyP0203OpsMag2.tyParam.tyNumPshrOffset.diValueMin 	:= -(tyP0203OpsMag2.tyOps.tyNumWidth.diValue/2 - p_tyMcParamCurr.diAWPusherAtHmPosInUM - IPshrSafeDistanceValue);
		tyP0203OpsMag2.tyParam.tyNumPshrOffset.diValueMax 	:= (tyP0203OpsMag2.tyOps.tyNumWidth.diValue/2 - p_tyMcParamCurr.diAWPusherAtHmPosInUM - IPshrSafeDistanceValue);
	ELSE
		tyP0203OpsMag2.tyParam.tyNumPshrOffset.diValueMin 	:= 0;
		tyP0203OpsMag2.tyParam.tyNumPshrOffset.diValueMax 	:= 0;
	END_IF

	//Control
	IF tyP0203OpsMag2.tyOps.tyBtnChgParam.bRtCompl = TRUE THEN
		tyP0203OpsMag2.tyOps.tyBtnChgParam.bRtCompl	:= FALSE;

		tyProdRcpCurrRcpWr	:= p_tyProdRcpCurrRcp0;

		tyP0203OpsMag2.tyParam.tyDrpDnMcMode.usiValueIdx	:= p_tyProdRcpCurrRcp0.usiMcMod;
		tyP0203OpsMag2.tyParam.tyNumMinSlt.diValue			:= p_tyProdRcpCurrRcp0.diMinSltValue;
		tyP0203OpsMag2.tyParam.tyNumMaxSlt.diValue			:= p_tyProdRcpCurrRcp0.diMaxSltValue;
		tyP0203OpsMag2.tyParam.tyNumPitch.diValue			:= p_tyProdRcpCurrRcp0.diPitch;
		tyP0203OpsMag2.tyParam.tyBtnToptoBtm.bValue			:= p_tyProdRcpCurrRcp0.bTopToBtm;
		tyP0203OpsMag2.tyParam.tyNumPshrExtSpeed.diValue 	:= p_tyProdRcpCurrRcp0.diMtrPshrExtSpd;
		tyP0203OpsMag2.tyParam.tyNumPshrExtTorque.diValue	:= p_tyProdRcpCurrRcp0.diMtrPshrExtTorq;
		tyP0203OpsMag2.tyParam.tyNumPshrOffset.diValue		:= p_tyProdRcpCurrRcp0.diPshrOffset;

		fUIInRtStatOff(ADR(tyP0203OpsMag2.tyParam.tyLyr.uiRtStat));

	END_IF

	tyP0203OpsMag2.tyOps.tyBtnChgParam.bValue		:= tyP0203OpsMag2.tyParam.tyLyr.uiRtStat.0 = FALSE;

	IF tyP0203OpsMag2.tyParam.tyLyr.uiRtStat.0 = FALSE THEN

		IF tyP0203OpsMag2.tyParam.tyBtnSave.bRtCompl = TRUE THEN

			tyProdRcpCurrRcpWr.usiMcMod			:= tyP0203OpsMag2.tyParam.tyDrpDnMcMode.usiValueIdx;
			tyProdRcpCurrRcpWr.diMinSltValue 	:= tyP0203OpsMag2.tyParam.tyNumMinSlt.diValue;
			tyProdRcpCurrRcpWr.diMaxSltValue 	:= tyP0203OpsMag2.tyParam.tyNumMaxSlt.diValue;
			tyProdRcpCurrRcpWr.diPitch 			:= tyP0203OpsMag2.tyParam.tyNumPitch.diValue;
			tyProdRcpCurrRcpWr.bTopToBtm 		:= tyP0203OpsMag2.tyParam.tyBtnToptoBtm.bValue;
			tyProdRcpCurrRcpWr.diMtrPshrExtSpd	:= tyP0203OpsMag2.tyParam.tyNumPshrExtSpeed.diValue;
			tyProdRcpCurrRcpWr.diMtrPshrExtTorq	:= tyP0203OpsMag2.tyParam.tyNumPshrExtTorque.diValue;
			tyProdRcpCurrRcpWr.diPshrOffset		:= tyP0203OpsMag2.tyParam.tyNumPshrOffset.diValue;

			eProdRcpAct	:= ProdRcpActWriteCurrRcpParam;

			IF p_eProdRcpStatus = Done AND p_eProdRcpStat = ProdRcpActWriteCurrRcpParam THEN
				eProdRcpAct	:= ProdRcpActIdle;

				//UIP0400
				tyP0400ProdSel.tyProdSel.tyTxtMcMode.usiValueIdx		:= p_tyProdRcpCurrRcp0.usiMcMod;
				tyP0400ProdSel.tyProdSel.tyNumMinSlt.diValue			:= p_tyProdRcpCurrRcp0.diMinSltValue;
				tyP0400ProdSel.tyProdSel.tyNumMaxSlt.diValue			:= p_tyProdRcpCurrRcp0.diMaxSltValue;
				tyP0400ProdSel.tyProdSel.tyNumPitch.diValue				:= p_tyProdRcpCurrRcp0.diPitch;
				tyP0400ProdSel.tyProdSel.tyBtnToptoBtm.bValue			:= p_tyProdRcpCurrRcp0.bTopToBtm;
				tyP0400ProdSel.tyProdSel.tyNumMtrPshrExtSpd.diValue		:= p_tyProdRcpCurrRcp0.diMtrPshrExtSpd;
				tyP0400ProdSel.tyProdSel.tyNumMtrPshrExtTorq.diValue	:= p_tyProdRcpCurrRcp0.diMtrPshrExtTorq;
				tyP0400ProdSel.tyProdSel.tyNumPshrOffset.diValue		:= p_tyProdRcpCurrRcp0.diPshrOffset;

				tyP0203OpsMag2.tyParam.tyBtnSave.bRtCompl			:= FALSE;
				tyP0203OpsMag2.tyParam.tyBtnSave.bValue				:= FALSE;

				fUIInRtStatHide(ADR(tyP0203OpsMag2.tyParam.tyLyr.uiRtStat));

			ELSIF p_eProdRcpStatus = Error THEN
				p_tyC0008MsgBox ACCESS ADR(tyP0203OpsMag2.tyMsgBoxSaveErr);

				IF tyP0203OpsMag2.tyMsgBoxSaveErr.tyBtnNo.bRtCompl = TRUE THEN
					tyP0203OpsMag2.tyMsgBoxSaveErr.tyBtnNo.bRtCompl	:= FALSE;
					tyP0203OpsMag2.tyMsgBoxSaveErr.tyBtnNo.bValue	:= FALSE;

					p_tyC0008MsgBox ACCESS ADR(tyP0203OpsMag2.tyMsgBoxHide);

					//Restore Param
					tyProdRcpCurrRcpWr	:= p_tyProdRcpCurrRcp2;

					tyP0203OpsMag2.tyParam.tyBtnSave.bRtCompl		:= FALSE;
					tyP0203OpsMag2.tyParam.tyBtnSave.bValue			:= FALSE;

					fUIInRtStatHide(ADR(tyP0203OpsMag2.tyParam.tyLyr.uiRtStat));

				END_IF

			END_IF

		ELSIF tyP0203OpsMag2.tyParam.tyBtnCancel.bRtCompl = TRUE THEN
			tyP0203OpsMag2.tyParam.tyBtnCancel.bRtCompl				:= FALSE;
			tyP0203OpsMag2.tyParam.tyBtnCancel.bValue				:= FALSE;

			fUIInRtStatHide(ADR(tyP0203OpsMag2.tyParam.tyLyr.uiRtStat));

		END_IF

	END_IF

	//Mask
	tyP0203OpsMag2.tyOps.tyBtnChgParam.uiMaskRtStat.0	:= p_tyUsrMgmtCurrAccessRgt.bChgParam AND p_bOpsStatusStop;

END_ACTION
```

#### Act_OptP0203InsertRmvMag.st
```iecst
ACTION Act_OptP0203InsertRmvMag:

	//Insert & Removed Magazine Manually Without Button Control
//	IF p_tyNtParamCurr.bProjBtnInsertRmvMag = FALSE THEN
//
//		IF p_bOpsStatusRun AND p_bOpsMagConvUL2InitDone THEN
//
//			fbMag2EntrySenOnTm(IN := p_tyDI.bMagConvEntSen2);
//
//			IF bNewMag2 = FALSE AND bRlsMag2 = FALSE THEN
//				IF p_bOpsMagConvUL2NewMagAllw AND fbMag2EntrySenOnTm.Q AND NOT p_bOpsMagConvUL2MagExitedWait THEN
//					bNewMag2	:= TRUE;
//				END_IF
//
//				IF p_bOpsMagConvUL2RlsMagAllw AND p_tyDI.bMagPresentSen2 AND p_tyDI.bOutShutterCloseRS AND p_tyBuffer2BffrStat.bBffrFull THEN
//					bRlsMag2	:= TRUE;
//				END_IF
//			END_IF
//
//			IF bNewMag2 = TRUE THEN
//
//				IF p_tyDI.bMag2FixedClampRS = TRUE AND p_tyDI.bMag2RemoteClampRS = TRUE THEN
//					bNewMag2	:= FALSE;
//				END_IF
//
//			ELSIF bRlsMag2 = TRUE THEN
//
//				IF p_tyDI.bMag2FixedUnclampRS = TRUE AND p_tyDI.bMag2RemoteUnclampRS = TRUE AND p_tyDI.bMagConvEntSen2 = TRUE THEN
//					bRlsMag2	:= FALSE;
//				END_IF
//
//			END_IF
//
//		ELSE
//
//			bNewMag2	:= FALSE;
//			bRlsMag2	:= FALSE;
//
//			fbMag2EntrySenOnTm(IN := FALSE);
//
//		END_IF
//
//	END_IF

END_ACTION
```

#### Act_OptP0203RstMnl.st
```iecst
ACTION Act_OptP0203RstMnl:

	IF eCurrPage <> UIP0203OpsMag2 AND eCurrPage <> UIP0003MMenu THEN
		bNewMag2	:= FALSE;
		bRlsMag2	:= FALSE;
		tyP0203OpsMag2.tyOps.tyBtnChgMag.bValue	:= FALSE;
		tyP0203OpsMag2.tyOps.tyBtnChgMag.bRtLk	:= FALSE;
		tyP0203OpsMag2.tyOps.tyBitmapChgMag.usiValueIdx	:= 0;

		tyP0003MMenu.tyMMenuBtn.tyBtnRlsNewMag2.bValue := FALSE;
		tyP0003MMenu.tyMMenuBtn.tyBtnRlsNewMag2.bRtLk  := FALSE;
		tyP0003MMenu.tyMMenuBtn.tyBtnRlsNewMag2.usiBitmapIdx := 0;
	END_IF

END_ACTION
```

#### Act_OptP0203Lane2ChgMag.st
```iecst
ACTION Act_OptP0203Lane2ChgMag:

	tyP0203OpsMag2.tyChgMag.tyBtnChgMag.bRtLk				:= FALSE;

	tChgMag ( IN:= tyP0203OpsMag2.tyChgMag.tyBtnChgMag.bValue = TRUE OR  FALSE , PT:=T#3s0ms);

	IF tChgMag.IN = TRUE THEN

	fbChgMagBlinkTm(IN := TRUE);

		IF fbChgMagBlinkTm.Q THEN
			fbChgMagBlinkTm(IN := FALSE);

			IF (tyP0203OpsMag2.tyChgMag.tyBitmapChgMag.usiValueIdx = 1) THEN
				tyP0203OpsMag2.tyChgMag.tyBitmapChgMag.usiValueIdx		:= 0;
			ELSE
				tyP0203OpsMag2.tyChgMag.tyBitmapChgMag.usiValueIdx		:= 1;
			END_IF
		END_IF
	ELSIF bChgMag = FALSE THEN

		tyP0203OpsMag2.tyChgMag.tyBitmapChgMag.usiValueIdx		:= 0;
	END_IF

	IF tChgMag.Q = TRUE THEN //(tyP0200OpsGen.tyChgMag.tyBtnChgMag.bRtCompl = TRUE) OR (tyP0203OpsMag2.tyChgMag.tyBtnChgMag.bRtCompl = TRUE)
	//	OR (tyP0203OpsMag2.tyChgMag.tyBtnChgMag.bRtCompl = TRUE)	OR (tyP0204OpsOutMagConv.tyChgMag.tyBtnChgMag.bRtCompl = TRUE) THEN

		tyP0203OpsMag2.tyChgMag.tyBitmapChgMag.usiValueIdx	:= 1;

		tyP0203OpsMag2.tyChgMag.tyBtnChgMag.bRtCompl			:= FALSE;

		bChgMag			:= TRUE;

//	ELSIF EDGEPOS(p_bFollower2SetBffrFull) THEN
//		bFllw2SetFull	:= TRUE;
//	ELSIF EDGEPOS(p_tyDI.bChgMagSig) THEN
//		bChgMagSig		:= TRUE;
	END_IF

	IF (p_bOpsOutMagConv2StepInitDone AND p_bOpsStatusRun = TRUE) AND bChgMag = TRUE THEN

		eBuffer2Act			:= BufferActSetFull;

		IF p_eBuffer2Stat = BufferActSetFull AND p_eBuffer2Status = Done THEN
			eBuffer1Act		:= BufferActIdle;

			bChgMag			:= FALSE;

		END_IF

//	ELSIF bFllw2SetFull = TRUE THEN
//		eBufferAct			:= BufferActSetFull;
//
//		IF p_eBufferStat = BufferActSetFull AND p_eBufferStatus = Done THEN
//			eBufferAct		:= BufferActIdle;
//
//			bFllw2SetFull	:= FALSE;
//		END_IF

	ELSIF (p_bOpsOutMagConv2StepInitDone AND p_bOpsStatusRun = TRUE) AND bChgMagSig THEN //ADAM Feature

		eBuffer2Act			:= BufferActSetFull;

		IF p_eBuffer2Stat = BufferActSetFull AND p_eBuffer2Status = Done THEN
			eBuffer2Act		:= BufferActIdle;

			bChgMagSig		:= FALSE;

		END_IF

	END_IF

	IF p_tyDI.bLifter2LmtSW = TRUE THEN
		fUIInRtStatHide(ADR(tyP0203OpsMag2.tyChgMag.tyBtnChgMag.uiMaskRtStat));
	ELSE
		fUIInRtStatOff(ADR(tyP0203OpsMag2.tyChgMag.tyBtnChgMag.uiMaskRtStat));
	END_IF

	//Manual unload magazine-------------------------------------------------------------------------------------------------------------
	IF p_bOpsRun THEN
		IF tyP0203OpsMag2.tyChgMag.tyBtnMnlUnloadMag.bValue THEN
			bOpsMnlUnloadMag2 := TRUE;
		ELSE
			bOpsMnlUnloadMag2 := FALSE;
		END_IF
	ELSE
		tyP0203OpsMag2.tyChgMag.tyBtnMnlUnloadMag.bValue := FALSE;
		bOpsMnlUnloadMag2 := FALSE;
	END_IF

	IF p_bOpsRun AND p_eOutMagConv2Status <> Busy THEN
		fUIInRtStatHide (ADR(tyP0203OpsMag2.tyChgMag.tyBtnMnlUnloadMag.uiMaskRtStat));
	ELSE
		fUIInRtStatOff (ADR(tyP0203OpsMag2.tyChgMag.tyBtnMnlUnloadMag.uiMaskRtStat));
	END_IF
END_ACTION
```

#### Act_OptP0203AIVDat.st - not listed in the package file held
```iecst
ACTION Act_OptP0203AIVDat:

	//Show Change Mag Button only in Manual Exchane Mode
	tyP0203OpsMag2.tyOps.tyBtnChgMag.uiRtStat.0 := p_tyMcParamCurr.eMagExMode = McSetMagXcAutoMode  AND p_tyMcParamCurr.eAGVComProtocol <> McSetAGVCommDisabled OR p_tyNtParamCurr.bProjLifterMagPlatform;
	tyP0203OpsMag2.tyOps.tyBitmapChgMag.uiRtStat.0 := p_tyMcParamCurr.eMagExMode = McSetMagXcAutoMode  AND p_tyMcParamCurr.eAGVComProtocol <> McSetAGVCommDisabled OR p_tyNtParamCurr.bProjLifterMagPlatform;

	//LED Wifi
	tyP0203OpsMag2.tyOps.tyBtnAIVWifi.bValue	:= p_bAGVOnline;

	//Change Magazine
	IF p_tyNtParamCurr.bProjBtnInsertRmvMag = TRUE THEN

		IF EDGENEG(p_bOpsStatusRun) THEN
			bNewMag2	:= FALSE;
			tyP0203OpsMag2.tyOps.tyBtnChgMag.bRtLk	:= FALSE;
			tyP0203OpsMag2.tyOps.tyBtnChgMag.bRtCompl	:= FALSE;
			tyP0203OpsMag2.tyOps.tyBtnChgMag.bValue		:= FALSE;
		END_IF

		IF tyP0203OpsMag2.tyOps.tyBtnChgMag.bRtCompl = TRUE THEN
			tyP0203OpsMag2.tyOps.tyBtnChgMag.bRtCompl	:= FALSE;
			bNewMag2	:= p_bOpsMagConvUL2NewMagAllw;
			bRlsMag2	:= p_bOpsMagConvUL2RlsMagAllw;
		END_IF

		IF bNewMag2 = TRUE THEN
			tyP0203OpsMag2.tyOps.tyBitmapChgMag.usiValueIdx	:= 1;
			IF p_tyDI.bMag2FixedUnclampRS = FALSE THEN
				bNewMag2	:= FALSE;
				tyP0203OpsMag2.tyOps.tyBtnChgMag.bValue	:= FALSE;
				tyP0203OpsMag2.tyOps.tyBtnChgMag.bRtLk	:= FALSE;
				tyP0203OpsMag2.tyOps.tyBitmapChgMag.usiValueIdx	:= 0;
			END_IF

		ELSIF bRlsMag2 = TRUE THEN
			tyP0203OpsMag2.tyOps.tyBitmapChgMag.usiValueIdx	:= 1;
			IF p_tyNtParamCurr.eCustomerReq = Siemens  THEN
				IF p_bOpsMagConvUL2EjectMESStep  THEN //FOR MES
					bRlsMag2	:= FALSE;
					tyP0203OpsMag2.tyOps.tyBtnChgMag.bValue	:= FALSE;
					tyP0203OpsMag2.tyOps.tyBtnChgMag.bRtLk	:= FALSE;
					tyP0203OpsMag2.tyOps.tyBitmapChgMag.usiValueIdx	:= 0;
				END_IF
			ELSIF p_tyDI.bMag2FixedUnclampRS = TRUE AND p_tyDI.bMagPresentSen2 = FALSE THEN
				bRlsMag2	:= FALSE;
				tyP0203OpsMag2.tyOps.tyBtnChgMag.bValue	:= FALSE;
				tyP0203OpsMag2.tyOps.tyBtnChgMag.bRtLk	:= FALSE;
				tyP0203OpsMag2.tyOps.tyBitmapChgMag.usiValueIdx	:= 0;
			END_IF

		ELSIF p_bAlarmErr THEN
			bNewMag2	:= FALSE;
			bRlsMag2	:= FALSE;
			tyP0203OpsMag2.tyOps.tyBtnChgMag.bValue	:= FALSE;
			tyP0203OpsMag2.tyOps.tyBtnChgMag.bRtLk	:= FALSE;
			tyP0203OpsMag2.tyOps.tyBitmapChgMag.usiValueIdx	:= 0;
		END_IF

		IF p_tyDI.bMagPresentSen2 AND p_tyDI.bMagConvEntSen2 = FALSE THEN
			tyP0203OpsMag2.tyOps.tyBtnChgMag.usiTxtIdx	:= 1;
		ELSE
			tyP0203OpsMag2.tyOps.tyBtnChgMag.usiTxtIdx	:= 0;
		END_IF

		IF (p_bOpsMagConvUL2NewMagAllw AND p_tyBuffer2BffrStat.bBffrMty)
			OR p_bOpsMagConvUL2RlsMagAllw
			OR p_bBufferMagRemoved2
			THEN //AND p_tyDI.bOutShutterCloseRS
			fUIInRtStatHide(ADR(tyP0203OpsMag2.tyOps.tyBtnChgMag.uiMaskRtStat));
		ELSE
			fUIInRtStatOff(ADR(tyP0203OpsMag2.tyOps.tyBtnChgMag.uiMaskRtStat));
		END_IF

	END_IF

END_ACTION
```

#### Act_EntP0204Disp.st
```iecst
ACTION Act_EntP0204Disp:

	//Access Address
	p_tyC0004Navi ACCESS ADR(tyP0204OpsMag3.tyNaviBack);

	p_tyC0005Main ACCESS ADR(tyCommon.tyMain);

	p_tyC0007Notif ACCESS ADR(tyCommon.tyNotif);

	p_tyC0008MsgBox ACCESS ADR(tyP0204OpsMag3.tyMsgBoxHide);

	p_tyC0009Info ACCESS ADR(tyCommon.tyInfo);

	p_tyC0011RcpPopUp ACCESS ADR(tyP0204OpsMag3.tyRcpPopUp);

	p_tyP0204Ops ACCESS ADR(tyP0204OpsMag3.tyOps);
	p_tyP0204IOMonitor ACCESS ADR(tyP0204OpsMag3.tyIOMonitor);
	p_tyP0204BypsInitConv ACCESS ADR(tyP0204OpsMag3.tyBypsInitConv);
	p_tyP0204Param ACCESS ADR(tyP0204OpsMag3.tyParam);

	//Display
	fUIInRtStatHide(ADR(tyP0204OpsMag3.tyIOMonitor.tyLyr.uiRtStat));
	fUIInRtStatHide(ADR(tyP0204OpsMag3.tyParam.tyLyr.uiRtStat));

	tyP0204OpsMag3.tyOps.tyBtnChgParam.uiRtStat.0	:= NOT(p_tyMcParamCurr.bChgParamEn);

	IF p_tyNtParamCurr.bMagAutoVerifyPrep = FALSE THEN
		tyP0204OpsMag3.tyIOMonitor.tyBtnMag3FixedClmpRS.usiTxtIdx	:= 44;
		tyP0204OpsMag3.tyIOMonitor.tyBtnMag3FixedUnclmpRS.usiTxtIdx:= 44;
		tyP0204OpsMag3.tyIOMonitor.tyBtnMag3RmtClmpRS.usiTxtIdx	:= 0;
		tyP0204OpsMag3.tyIOMonitor.tyBtnMag3RmtUnclmpRS.usiTxtIdx:= 0;
		tyP0204OpsMag3.tyIOMonitor.tyBtnMag3FixedClampCtrl.usiTxtIdx:= 34;
		tyP0204OpsMag3.tyIOMonitor.tyBtnMag3RemoteClampCtrl.usiTxtIdx:= 0;
	ELSE
		//	tyP0204OpsMag3.tyIOMonitor.tyBtnMag3FixedClmpRS.usiTxtIdx	:= 74;
		tyP0204OpsMag3.tyIOMonitor.tyBtnMag3FixedUnclmpRS.usiTxtIdx:= 44;
		//	tyP0204OpsMag3.tyIOMonitor.tyBtnMag3RmtClmpRS.usiTxtIdx	:= 51;
		//	tyP0204OpsMag3.tyIOMonitor.tyBtnMag3RmtUnclmpRS.usiTxtIdx:= 50;
			tyP0204OpsMag3.tyIOMonitor.tyBtnMag3FixedClampCtrl.usiTxtIdx:= 34;
		//	tyP0204OpsMag3.tyIOMonitor.tyBtnMag3RemoteClampCtrl.usiTxtIdx:= 19;

	END_IF

	tyP0204OpsMag3.tyParam.tyNumMaxSlt.diValueMax	:= p_tyMagRcpCurrRcp.diTtlSlt;

END_ACTION
```

#### Act_OptP0204Navi.st
```iecst
ACTION Act_OptP0204Navi:

	IF tyP0204OpsMag3.tyNaviBack.tyBtnBack.bRtCompl = TRUE THEN
		tyP0204OpsMag3.tyNaviBack.tyBtnBack.bRtCompl	:= FALSE;
		tyP0204OpsMag3.tyNaviBack.tyBtnBack.bValue		:= FALSE;

		eChgPage	:= UIP0200OpsGen;

	END_IF

END_ACTION
```

#### Act_OptP0204ChgPage.st
```iecst
ACTION Act_OptP0204ChgPage:

	IF tyP0204OpsMag3.tyOps.tyHotspotMagInfo.bRtCompl = TRUE THEN
		tyP0204OpsMag3.tyOps.tyHotspotMagInfo.bRtCompl	:= FALSE;

		eChgPage	:= UIP0800MagInfo;
	END_IF

END_ACTION
```

#### Act_OptP0204UpdtDat.st
```iecst
ACTION Act_OptP0204UpdtDat:

	//Status
	fbMcStatUpdtTm(IN := TRUE);
	IF fbMcStatUpdtTm.Q = TRUE THEN
		fbMcStatUpdtTm(IN := FALSE);

//		IF p_tyNtParamCurr.bProjMag3ConvPrep = FALSE THEN
//			tyP0204OpsMag3.tyOps.tyStringMcStat.sValue	:= p_sOpsMagUL3StepTxt;
//		ELSE
//			tyP0204OpsMag3.tyOps.tyStringMcStat.sValue	:= p_sOpsMagConvUL3StepTxt;
//		END_IF

		IF p_tyNtParamCurr.bProjLifterMagPlatform THEN
			tyP0204OpsMag3.tyOps.tyStringMcStat.sValue		:= p_sOpsLifMagULStepTxt;
		ELSE
			tyP0204OpsMag3.tyOps.tyStringMcStat.sValue	:= p_sOpsMagConvUL3StepTxt;
		END_IF

	END_IF

	//Conveyor Auto Width
	IF p_tyNtParamCurr.bAWPrep = TRUE AND p_tyMcParamCurr.bAWDis = FALSE THEN
		tyP0204OpsMag3.tyOps.tyNumWidth.diValue		:= p_tyMcParamCurr.diWidthAtHmPosInUM - p_diAWOpenActualPos;
		tyP0204OpsMag3.tyOps.tyNumWidth2.diValue	:= p_tyMcParamCurr.diWidthAtHmPosInUM - p_diAWOpenActualPos;
	ELSE
		tyP0204OpsMag3.tyOps.tyNumWidth.diValue		:= p_tyProdRcpCurrRcp1.diWidthInUM;
		tyP0204OpsMag3.tyOps.tyNumWidth2.diValue		:= p_tyProdRcpCurrRcp1.diWidthInUM2;
	END_IF

	//Program Info

	IF p_bMcParamAutoRcpDisable OR p_bNtParamAutoRcpF1ArbitraryType  THEN
		tyP0204OpsMag3.tyOps.tyTxtMod.usiValueIdx	:= p_tyProdRcpCurrRcp2.usiMcMod;
		tyP0204OpsMag3.tyOps.tyNumMinSltRange.diValue	:= p_tyProdRcpCurrRcp2.diMinSltValue;
		tyP0204OpsMag3.tyOps.tyNumMaxSltRange.diValue	:= p_tyProdRcpCurrRcp2.diMaxSltValue;
		tyP0204OpsMag3.tyOps.tyBtnToptoBtm.bValue		:= p_tyProdRcpCurrRcp2.bTopToBtm;
		tyP0204OpsMag3.tyOps.tyNumPitch.diValue			:= p_tyProdRcpCurrRcp2.diPitch;
		tyP0204OpsMag3.tyOps.tyStringProdNm.sValue		:= p_tyProdRcpCurrRcp2.sRcpNm;
	ELSE  //FALSE AutoRcp Mode
		tyP0204OpsMag3.tyOps.tyTxtMod.usiValueIdx	:= p_tyProdRcpCurrRcp0.usiMcMod;

		tyP0204OpsMag3.tyOps.tyNumMinSltRange.diValue	:= pa_tyMagProps[3].diMinSlt;
		tyP0204OpsMag3.tyOps.tyNumMaxSltRange.diValue	:= pa_tyMagProps[3].diMaxSlt;
		tyP0204OpsMag3.tyOps.tyBtnToptoBtm.bValue		:= p_tyProdRcpCurrRcp0.bTopToBtm;
		tyP0204OpsMag3.tyOps.tyNumPitch.diValue			:= pa_tyMagProps[3].diPitch;
		IF p_tyNtParamCurr.eAutoRcpPrecededBy =  PrecededBySelf THEN
			tyP0204OpsMag3.tyOps.tyStringProdNm.sValue		:= pa_tyAutoRcpBrdProps[3].sProductTypeId;
		ELSIF p_tyNtParamCurr.eAutoRcpPrecededBy =  PrecededByF1 THEN
			tyP0204OpsMag3.tyOps.tyStringProdNm.sValue		:= pa_tyMagProps[3].sRcpNm;
		END_IF
	END_IF
	//Magazine Info
	tyP0204OpsMag3.tyOps.tyStringMagNm.sValue	:= p_tyMagRcpCurrRcp.sRcpNm;

	IF p_bBuffer3MagPresent = TRUE THEN
		IF p_tyNtParamCurr.eCustomerReq = Siemens AND p_iOpsMagConvUL3MESAcptCond <= 0 AND  p_tyMcParamCurr.bMESEn THEN
			tyP0204OpsMag3.tyOps.tyNumMag3AvlQty.diValue	:= 0;
			tyP0204OpsMag3.tyOps.tyNumMag3TtlSlt.diValue	:= 0;
		ELSE
			tyP0204OpsMag3.tyOps.tyNumMag3AvlQty.diValue	:= p_tyBuffer3BffrStat.diTtlBrdCap - (p_tyBuffer3BffrStat.diTtlGdBrd + p_tyBuffer3BffrStat.diTtlBadBrd);
			tyP0204OpsMag3.tyOps.tyNumMag3TtlSlt.diValue	:= p_tyBuffer3BffrStat.diTtlBrdCap;
		END_IF
	ELSE
		tyP0204OpsMag3.tyOps.tyNumMag3AvlQty.diValue	:= 0;
		tyP0204OpsMag3.tyOps.tyNumMag3TtlSlt.diValue	:= 0;
	END_IF

	//Magazine Present States
	IF p_bBuffer3MagPresent = TRUE THEN

		IF p_tyBuffer3BffrStat.bBffrFull = TRUE THEN
			tyP0204OpsMag3.tyOps.tyTxtMag3Stat.usiValueIdx := 2;
			tyP0204OpsMag3.tyOps.tyTxtMag3Stat.usiColor	   := 1;
		ELSIF p_tyBuffer3BffrStat.bBffrMty = TRUE THEN
			tyP0204OpsMag3.tyOps.tyTxtMag3Stat.usiValueIdx := 1;
			tyP0204OpsMag3.tyOps.tyTxtMag3Stat.usiColor	   := 0;
		ELSE
			tyP0204OpsMag3.tyOps.tyTxtMag3Stat.usiValueIdx := 3;
			tyP0204OpsMag3.tyOps.tyTxtMag3Stat.usiColor	   := 0;
		END_IF

	ELSE
		tyP0204OpsMag3.tyOps.tyTxtMag3Stat.usiValueIdx := 0;
		tyP0204OpsMag3.tyOps.tyTxtMag3Stat.usiColor	   := 1;
	END_IF

	//Product Recipe 254
	tyP0204OpsMag3.tyOps.tyHotspotShowLRcp.uiRtStat.0 := NOT(tyP0204OpsMag3.tyOps.tyStringProdNm.sValue <> '');

	IF tyP0204OpsMag3.tyOps.tyHotspotShowLRcp.bRtCompl = TRUE THEN
		tyP0204OpsMag3.tyOps.tyHotspotShowLRcp.bRtCompl := FALSE;

		fUIInRtStatOff(ADR(tyP0204OpsMag3.tyRcpPopUp.tyLyr.uiRtStat));

		tyP0204OpsMag3.tyRcpPopUp.tyStringInfo.sValue  := p_tyProdRcpCurrRcp1.sRcpNm;

	ELSIF tyP0204OpsMag3.tyRcpPopUp.tyHotspotClose.bRtCompl = TRUE THEN
		tyP0204OpsMag3.tyRcpPopUp.tyHotspotClose.bRtCompl := FALSE;

		fUIInRtStatHide(ADR(tyP0204OpsMag3.tyRcpPopUp.tyLyr.uiRtStat));

	END_IF

END_ACTION
```

#### Act_OptP0204IOMonitor.st
```iecst
ACTION Act_OptP0204IOMonitor:

	IF tyP0204OpsMag3.tyOps.tyHotspotIOMonitor.bRtCompl = TRUE THEN
		tyP0204OpsMag3.tyOps.tyHotspotIOMonitor.bRtCompl	:= FALSE;

		fUIInRtStatOff(ADR(tyP0204OpsMag3.tyIOMonitor.tyLyr.uiRtStat));

		p_tyC0004Navi ACCESS ADR(tyP0204OpsMag3.tyNaviHide);

	ELSIF tyP0204OpsMag3.tyIOMonitor.tyHotspotClose.bRtCompl = TRUE THEN
		tyP0204OpsMag3.tyIOMonitor.tyHotspotClose.bRtCompl	:= FALSE;

		fUIInRtStatHide(ADR(tyP0204OpsMag3.tyIOMonitor.tyLyr.uiRtStat));

		p_tyC0004Navi ACCESS ADR(tyP0204OpsMag3.tyNaviBack);

	END_IF

	IF tyP0204OpsMag3.tyIOMonitor.tyLyr.uiRtStat.0 = FALSE THEN

		//Digital Input
		tyP0204OpsMag3.tyIOMonitor.tyBtnSafetyRlySig.bValue				:= p_tyDI.bSafetyRlySig;
		tyP0204OpsMag3.tyIOMonitor.tyBtnEStop.bValue					:= p_tyDI.bEStopSig;
		tyP0204OpsMag3.tyIOMonitor.tyBtnCoverSWSig.bValue				:= p_tyDI.bCoverSWSig;
		tyP0204OpsMag3.tyIOMonitor.tyBtnUBAA.bValue						:= p_tyDI.bUBAA;
		tyP0204OpsMag3.tyIOMonitor.tyBtnUBAB.bValue						:= p_tyDI.bUBAB;
		tyP0204OpsMag3.tyIOMonitor.tyBtnUBAAStat.bValue					:= p_tyDI.bUBAAStat;
		tyP0204OpsMag3.tyIOMonitor.tyBtnUBABStat.bValue					:= p_tyDI.bUBABStat;
		tyP0204OpsMag3.tyIOMonitor.tyBtnOvenInfeedSigA.bValue			:= p_tyDI.bOvenInfeedSigA;
		tyP0204OpsMag3.tyIOMonitor.tyBtnOvenInfeedSigB.bValue			:= p_tyDI.bOvenInfeedSigB;
		tyP0204OpsMag3.tyIOMonitor.tyBtnMag3FixedClmpRS.bValue			:= p_tyDI.bMag3FixedClampRS;
		tyP0204OpsMag3.tyIOMonitor.tyBtnMag3FixedUnclmpRS.bValue		:= p_tyDI.bMag3FixedUnclampRS;
		tyP0204OpsMag3.tyIOMonitor.tyBtnMag3RmtClmpRS.bValue			:= p_tyDI.bMag3RemoteClampRS;
		tyP0204OpsMag3.tyIOMonitor.tyBtnMag3RmtUnclmpRS.bValue			:= p_tyDI.bMag3RemoteUnclampRS;
		tyP0204OpsMag3.tyIOMonitor.tyBtnMag3ConvEntrySen.bValue			:= p_tyDI.bMagConvEntSen3;
		tyP0204OpsMag3.tyIOMonitor.tyBtnMag3PresentSen.bValue			:= p_tyDI.bMagPresentSen3;
		tyP0204OpsMag3.tyIOMonitor.tyBtnMag3AIVInPosSen1.bValue			:= p_tyDI.bMag3AIVInPosSen1;
		tyP0204OpsMag3.tyIOMonitor.tyBtnMag3AIVInPosSen2.bValue			:= p_tyDI.bMag3AIVInPosSen2;
		tyP0204OpsMag3.tyIOMonitor.tyBtnMag3OrientationChkSen1.bValue	:= p_tyDI.bMag3OrientChkSen1;
		tyP0204OpsMag3.tyIOMonitor.tyBtnMag3OrientationChkSen2.bValue	:= p_tyDI.bMag3OrientChkSen2;

		tyP0204OpsMag3.tyIOMonitor.tyBtnSelUnclampRS.bValue				:= p_tyDI.bMag3SelUnClampRS;

		tyP0204OpsMag3.tyIOMonitor.tyBtnCAB717Sen.bValue				:= p_tyDI.bMagConvCAB717MagSen3;
//		tyP0204OpsMag3.tyIOMonitor.tyBtnHeightSen.bValue				:= p_tyDI.bMagConvHeightSen3;
		tyP0204OpsMag3.tyIOMonitor.tyBtnMagSmallSen.bValue				:= p_tyDI.bMagConvSmallMagSen3;
		tyP0204OpsMag3.tyIOMonitor.tyBtnMagLargeSen.bValue				:= p_tyDI.bMagConvLargeMagSen3;
		tyP0204OpsMag3.tyIOMonitor.tyBtnCurtainSen.bValue				:= p_tyDI.bCurtainSen;
		tyP0204OpsMag3.tyIOMonitor.tyBtnCurtainSenPB.bValue				:= p_tyDI.bCurtainSenPB;
		tyP0204OpsMag3.tyIOMonitor.tyBtnMag3DetSen.bValue				:= p_tyDI.bMag3FixedClampSen;

		//MagHeightCheckSensor
		IF p_tyNtParamCurr.bMagAutoVerifyPrep = TRUE THEN
			tyP0204OpsMag3.tyIOMonitor.tyBtnHeightSen.bValue			:= p_tyDI.bMagConvHeightSen3;
		ELSE
			tyP0204OpsMag3.tyIOMonitor.tyBtnHeightSen.bValue			:= p_tyDI.bHighMagDetSen3;
		END_IF

		//Digital Output
		tyP0204OpsMag3.tyIOMonitor.tyBtnSafetyRlyRst.bValue				:= p_tyDO.bSafetyRlyRst;
		tyP0204OpsMag3.tyIOMonitor.tyBtnTLGreen.bValue					:= p_tyDO.bTLGreen;
		tyP0204OpsMag3.tyIOMonitor.tyBtnTLAmber.bValue					:= p_tyDO.bTLAmber;
		tyP0204OpsMag3.tyIOMonitor.tyBtnTLRed.bValue					:= p_tyDO.bTLRed;
		tyP0204OpsMag3.tyIOMonitor.tyBtnBuzzer.bValue					:= p_tyDO.bBuzzer;
		tyP0204OpsMag3.tyIOMonitor.tyBtnUSBA.bValue						:= p_tyDO.bUSBA;
		tyP0204OpsMag3.tyIOMonitor.tyBtnUSBB.bValue						:= p_tyDO.bUSBB;
		tyP0204OpsMag3.tyIOMonitor.tyBtnOvenInfoSigA.bValue				:= p_tyDO.bOvenInfoSigA;
		tyP0204OpsMag3.tyIOMonitor.tyBtnOvenInfoSigB.bValue				:= p_tyDO.bOvenInfoSigB;
		tyP0204OpsMag3.tyIOMonitor.tyBtnMag3FixedClampCtrl.bValue		:= p_tyDO.bMag3FixedClampCtrl;
		tyP0204OpsMag3.tyIOMonitor.tyBtnMag3RemoteClampCtrl.bValue		:= p_tyDO.bMag3RemoteClampCtrl;
		tyP0204OpsMag3.tyIOMonitor.tyBtnMag3ConvMtrIn.bValue			:= p_tyDO.bMag3ConvMtrIn;
		tyP0204OpsMag3.tyIOMonitor.tyBtnMag3ConvMtrOut.bValue			:= p_tyDO.bMag3ConvMtrOut;
		tyP0204OpsMag3.tyIOMonitor.tyBtnMagSelClampCtrl.bValue			:= p_tyDO.bMag3SelClampCtrl;
		//tyP0204OpsMag3.tyIOMonitor.tyBtnMagSelUnClampCtrl.bValue		:= p_tyDO.bMag3SelUnClampCtrl;
		tyP0204OpsMag3.tyIOMonitor.tyBtnCurtainSenPBLED.bValue			:= p_tyDO.bBypCurtainPBLED;
	END_IF

END_ACTION
```

#### Act_OptP0204_P0003AIVDat.st
```iecst
ACTION Act_OptP0204_P0003AIVDat:

	//Show Change Mag Button only in Manual Exchane Mode
	tyP0204OpsMag3.tyOps.tyBtnChgMag.uiRtStat.0 := p_tyMcParamCurr.eMagExMode = McSetMagXcAutoMode AND p_tyMcParamCurr.eAGVComProtocol <> McSetAGVCommDisabled OR p_tyNtParamCurr.bProjLifterMagPlatform;
	tyP0204OpsMag3.tyOps.tyBitmapChgMag.uiRtStat.0 := p_tyMcParamCurr.eMagExMode = McSetMagXcAutoMode AND p_tyMcParamCurr.eAGVComProtocol <> McSetAGVCommDisabled OR p_tyNtParamCurr.bProjLifterMagPlatform;

	//LED Wifi
	tyP0204OpsMag3.tyOps.tyBtnAIVWifi.bValue	:= p_bAGVOnline;

	//Change Magazine
	IF p_tyNtParamCurr.bProjBtnInsertRmvMag = TRUE THEN

		IF EDGENEG(p_bOpsStatusRun) THEN
			bNewMag3	:= FALSE;
			tyP0204OpsMag3.tyOps.tyBtnChgMag.bRtLk	:= FALSE;
			tyP0204OpsMag3.tyOps.tyBtnChgMag.bRtCompl	:= FALSE;
			tyP0003MMenu.tyMMenuBtn.tyBtnRlsNewMag3.bRtLk := FALSE;
			tyP0003MMenu.tyMMenuBtn.tyBtnRlsNewMag3.bRtCompl := FALSE;
			tyP0204OpsMag3.tyOps.tyBtnChgMag.bValue		:= FALSE;
			tyP0003MMenu.tyMMenuBtn.tyBtnRlsNewMag3.bValue := FALSE;
		END_IF

		IF tyP0204OpsMag3.tyOps.tyBtnChgMag.bRtCompl = TRUE OR tyP0003MMenu.tyMMenuBtn.tyBtnRlsNewMag3.bRtCompl THEN
			tyP0204OpsMag3.tyOps.tyBtnChgMag.bRtCompl	:= FALSE;
			tyP0003MMenu.tyMMenuBtn.tyBtnRlsNewMag3.bRtCompl := FALSE;
			bNewMag3	:= p_bOpsMagConvUL3NewMagAllw;
			bRlsMag3	:= p_bOpsMagConvUL3RlsMagAllw;
		END_IF

		IF bNewMag3 = TRUE THEN
			tyP0204OpsMag3.tyOps.tyBitmapChgMag.usiValueIdx	:= 1;
			tyP0003MMenu.tyMMenuBtn.tyBtnRlsNewMag3.usiBitmapIdx := 1;
			IF p_tyDI.bMag3FixedUnclampRS = FALSE THEN
				bNewMag3	:= FALSE;
				tyP0204OpsMag3.tyOps.tyBtnChgMag.bValue	:= FALSE;
				tyP0003MMenu.tyMMenuBtn.tyBtnRlsNewMag3.bValue := FALSE;
				tyP0204OpsMag3.tyOps.tyBtnChgMag.bRtLk	:= FALSE;
				tyP0003MMenu.tyMMenuBtn.tyBtnRlsNewMag3.bRtLk := FALSE;
				tyP0204OpsMag3.tyOps.tyBitmapChgMag.usiValueIdx	:= 0;
				tyP0003MMenu.tyMMenuBtn.tyBtnRlsNewMag3.usiBitmapIdx := 0;
			END_IF

		ELSIF bRlsMag3 = TRUE THEN
			tyP0204OpsMag3.tyOps.tyBitmapChgMag.usiValueIdx	:= 1;
			tyP0003MMenu.tyMMenuBtn.tyBtnRlsNewMag3.usiBitmapIdx := 1;
			IF p_tyNtParamCurr.eCustomerReq = Siemens THEN
				IF p_bOpsMagConvUL3EjectMESStep  THEN //FOR MES
					bRlsMag3	:= FALSE;
					tyP0204OpsMag3.tyOps.tyBtnChgMag.bValue	:= FALSE;
					tyP0003MMenu.tyMMenuBtn.tyBtnRlsNewMag3.bValue := FALSE;
					tyP0204OpsMag3.tyOps.tyBtnChgMag.bRtLk	:= FALSE;
					tyP0003MMenu.tyMMenuBtn.tyBtnRlsNewMag3.bRtLk := FALSE;
					tyP0204OpsMag3.tyOps.tyBitmapChgMag.usiValueIdx	:= 0;
					tyP0003MMenu.tyMMenuBtn.tyBtnRlsNewMag3.usiBitmapIdx := 0;
				END_IF
			ELSIF (p_tyDI.bMag3FixedUnclampRS = TRUE AND p_tyDI.bMagPresentSen3 = FALSE) THEN
				bRlsMag3	:= FALSE;
				tyP0204OpsMag3.tyOps.tyBtnChgMag.bValue	:= FALSE;
				tyP0003MMenu.tyMMenuBtn.tyBtnRlsNewMag3.bValue := FALSE;
				tyP0204OpsMag3.tyOps.tyBtnChgMag.bRtLk	:= FALSE;
				tyP0003MMenu.tyMMenuBtn.tyBtnRlsNewMag3.bRtLk := FALSE;
				tyP0204OpsMag3.tyOps.tyBitmapChgMag.usiValueIdx	:= 0;
				tyP0003MMenu.tyMMenuBtn.tyBtnRlsNewMag3.usiBitmapIdx := 0;
			END_IF

		ELSIF p_bAlarmErr THEN
			bNewMag3	:= FALSE;
			bRlsMag3	:= FALSE;
			tyP0204OpsMag3.tyOps.tyBtnChgMag.bValue	:= FALSE;
			tyP0003MMenu.tyMMenuBtn.tyBtnRlsNewMag3.bValue := FALSE;
			tyP0204OpsMag3.tyOps.tyBtnChgMag.bRtLk	:= FALSE;
			tyP0003MMenu.tyMMenuBtn.tyBtnRlsNewMag3.bRtLk:= FALSE;
			tyP0204OpsMag3.tyOps.tyBitmapChgMag.usiValueIdx	:= 0;
			tyP0003MMenu.tyMMenuBtn.tyBtnRlsNewMag3.usiBitmapIdx := 0;
		END_IF

		IF p_tyDI.bMagPresentSen3 AND p_tyDI.bMagConvEntSen3 = FALSE THEN
			tyP0204OpsMag3.tyOps.tyBtnChgMag.usiTxtIdx	:= 1;
			tyP0003MMenu.tyMMenuBtn.tyBtnRlsNewMag3.usiTxtIdx := 33;
		ELSE
			tyP0204OpsMag3.tyOps.tyBtnChgMag.usiTxtIdx	:= 0;
			tyP0003MMenu.tyMMenuBtn.tyBtnRlsNewMag3.usiTxtIdx := 8;
		END_IF

		IF (p_bOpsMagConvUL3NewMagAllw AND p_tyBuffer3BffrStat.bBffrMty)
			OR p_bOpsMagConvUL3RlsMagAllw
			OR p_bBufferMagRemoved3
			THEN //AND p_tyDI.bOutShutterCloseRS
			fUIInRtStatHide(ADR(tyP0204OpsMag3.tyOps.tyBtnChgMag.uiMaskRtStat));
			fUIInRtStatHide(ADR(tyP0003MMenu.tyMMenuBtn.tyBtnRlsNewMag3.uiMaskRtStat));
		ELSE
			fUIInRtStatOff(ADR(tyP0204OpsMag3.tyOps.tyBtnChgMag.uiMaskRtStat));
			fUIInRtStatOff(ADR(tyP0003MMenu.tyMMenuBtn.tyBtnRlsNewMag3.uiMaskRtStat));
		END_IF

	END_IF

END_ACTION
```

#### Act_OptP0204ChgParam.st
```iecst
ACTION Act_OptP0204ChgParam:

	tyP0204OpsMag3.tyParam.tyNumMinSlt.diValueMax		:= tyP0204OpsMag3.tyParam.tyNumMaxSlt.diValue;
	tyP0204OpsMag3.tyParam.tyNumMaxSlt.diValueMin		:= tyP0204OpsMag3.tyParam.tyNumMinSlt.diValue;
	tyP0204OpsMag3.tyParam.tyNumPitch.diValueMax		:= tyP0204OpsMag3.tyParam.tyNumMaxSlt.diValue - tyP0204OpsMag3.tyParam.tyNumMinSlt.diValue + 1;
	tyP0204OpsMag3.tyParam.tyNumPitch.diValueMin		:= 1;
	tyP0204OpsMag3.tyOps.tyBtnChgParam.uiRtStat.0	:= NOT(p_tyMcParamCurr.bChgParamEn);

	tyP0204OpsMag3.tyParam.tyNumPshrExtSpeed.diValueMin 	:= p_tyNtParamCurr.tyProdRcpMtrPshrExtSpd.diMin;
	tyP0204OpsMag3.tyParam.tyNumPshrExtSpeed.diValueMax 	:= p_tyNtParamCurr.tyProdRcpMtrPshrExtSpd.diMax;
	tyP0204OpsMag3.tyParam.tyNumPshrExtTorque.diValueMin	:= p_tyNtParamCurr.tyProdRcpMtrPshrExtTorq.diMin;
	tyP0204OpsMag3.tyParam.tyNumPshrExtTorque.diValueMax	:= p_tyNtParamCurr.tyProdRcpMtrPshrExtTorq.diMax;
	tyP0204OpsMag3.tyParam.tyNumPshrExtSpeed.uiRtStat.0		:= NOT p_tyNtParamCurr.bProjMotorizedPusherPrep;
	tyP0204OpsMag3.tyParam.tyNumPshrExtTorque.uiRtStat.0	:= NOT p_tyNtParamCurr.bProjMotorizedPusherPrep;

	IF (tyP0204OpsMag3.tyOps.tyNumWidth.diValue) <> 0 THEN
		tyP0204OpsMag3.tyParam.tyNumPshrOffset.diValueMin 	:= -(tyP0204OpsMag3.tyOps.tyNumWidth.diValue/2 - p_tyMcParamCurr.diAWPusherAtHmPosInUM - IPshrSafeDistanceValue);
		tyP0204OpsMag3.tyParam.tyNumPshrOffset.diValueMax 	:= (tyP0204OpsMag3.tyOps.tyNumWidth.diValue/2 - p_tyMcParamCurr.diAWPusherAtHmPosInUM - IPshrSafeDistanceValue);
	ELSE
		tyP0204OpsMag3.tyParam.tyNumPshrOffset.diValueMin 	:= 0;
		tyP0204OpsMag3.tyParam.tyNumPshrOffset.diValueMax 	:= 0;
	END_IF

	//Control
	IF tyP0204OpsMag3.tyOps.tyBtnChgParam.bRtCompl = TRUE THEN
		tyP0204OpsMag3.tyOps.tyBtnChgParam.bRtCompl	:= FALSE;

		tyProdRcpCurrRcpWr	:= p_tyProdRcpCurrRcp0;

		tyP0204OpsMag3.tyParam.tyDrpDnMcMode.usiValueIdx	:= p_tyProdRcpCurrRcp0.usiMcMod;
		tyP0204OpsMag3.tyParam.tyNumMinSlt.diValue	:= p_tyProdRcpCurrRcp0.diMinSltValue;
		tyP0204OpsMag3.tyParam.tyNumMaxSlt.diValue	:= p_tyProdRcpCurrRcp0.diMaxSltValue;
		tyP0204OpsMag3.tyParam.tyNumPitch.diValue		:= p_tyProdRcpCurrRcp0.diPitch;
		tyP0204OpsMag3.tyParam.tyBtnToptoBtm.bValue	:= p_tyProdRcpCurrRcp0.bTopToBtm;
		tyP0204OpsMag3.tyParam.tyNumPshrExtSpeed.diValue 	:= p_tyProdRcpCurrRcp0.diMtrPshrExtSpd;
		tyP0204OpsMag3.tyParam.tyNumPshrExtTorque.diValue	:= p_tyProdRcpCurrRcp0.diMtrPshrExtTorq;
		tyP0204OpsMag3.tyParam.tyNumPshrOffset.diValue		:= p_tyProdRcpCurrRcp0.diPshrOffset;

		fUIInRtStatOff(ADR(tyP0204OpsMag3.tyParam.tyLyr.uiRtStat));

	END_IF

	tyP0204OpsMag3.tyOps.tyBtnChgParam.bValue	:= tyP0204OpsMag3.tyParam.tyLyr.uiRtStat.0 = FALSE;

	IF tyP0204OpsMag3.tyParam.tyLyr.uiRtStat.0 = FALSE THEN

		IF tyP0204OpsMag3.tyParam.tyBtnSave.bRtCompl = TRUE THEN

			tyProdRcpCurrRcpWr.usiMcMod			:= tyP0204OpsMag3.tyParam.tyDrpDnMcMode.usiValueIdx;
			tyProdRcpCurrRcpWr.diMinSltValue 	:= tyP0204OpsMag3.tyParam.tyNumMinSlt.diValue;
			tyProdRcpCurrRcpWr.diMaxSltValue 	:= tyP0204OpsMag3.tyParam.tyNumMaxSlt.diValue;
			tyProdRcpCurrRcpWr.diPitch 			:= tyP0204OpsMag3.tyParam.tyNumPitch.diValue;
			tyProdRcpCurrRcpWr.bTopToBtm 		:= tyP0204OpsMag3.tyParam.tyBtnToptoBtm.bValue;
			tyProdRcpCurrRcpWr.diMtrPshrExtSpd	:= tyP0204OpsMag3.tyParam.tyNumPshrExtSpeed.diValue;
			tyProdRcpCurrRcpWr.diMtrPshrExtTorq	:= tyP0204OpsMag3.tyParam.tyNumPshrExtTorque.diValue;
			tyProdRcpCurrRcpWr.diPshrOffset		:= tyP0204OpsMag3.tyParam.tyNumPshrOffset.diValue;

			eProdRcpAct	:= ProdRcpActWriteCurrRcpParam;

			IF p_eProdRcpStatus = Done AND p_eProdRcpStat = ProdRcpActWriteCurrRcpParam THEN
				eProdRcpAct	:= ProdRcpActIdle;

				//UIP0400
				tyP0400ProdSel.tyProdSel.tyTxtMcMode.usiValueIdx		:= p_tyProdRcpCurrRcp0.usiMcMod;
				tyP0400ProdSel.tyProdSel.tyNumMinSlt.diValue			:= p_tyProdRcpCurrRcp0.diMinSltValue;
				tyP0400ProdSel.tyProdSel.tyNumMaxSlt.diValue			:= p_tyProdRcpCurrRcp0.diMaxSltValue;
				tyP0400ProdSel.tyProdSel.tyNumPitch.diValue				:= p_tyProdRcpCurrRcp0.diPitch;
				tyP0400ProdSel.tyProdSel.tyBtnToptoBtm.bValue			:= p_tyProdRcpCurrRcp0.bTopToBtm;
				tyP0400ProdSel.tyProdSel.tyNumMtrPshrExtSpd.diValue		:= p_tyProdRcpCurrRcp0.diMtrPshrExtSpd;
				tyP0400ProdSel.tyProdSel.tyNumMtrPshrExtTorq.diValue	:= p_tyProdRcpCurrRcp0.diMtrPshrExtTorq;
				tyP0400ProdSel.tyProdSel.tyNumPshrOffset.diValue		:= p_tyProdRcpCurrRcp0.diPshrOffset;

				tyP0204OpsMag3.tyParam.tyBtnSave.bRtCompl	:= FALSE;
				tyP0204OpsMag3.tyParam.tyBtnSave.bValue		:= FALSE;

				fUIInRtStatHide(ADR(tyP0204OpsMag3.tyParam.tyLyr.uiRtStat));

			ELSIF p_eProdRcpStatus = Error THEN
				p_tyC0008MsgBox ACCESS ADR(tyP0204OpsMag3.tyMsgBoxSaveErr);

				IF tyP0204OpsMag3.tyMsgBoxSaveErr.tyBtnNo.bRtCompl = TRUE THEN
					tyP0204OpsMag3.tyMsgBoxSaveErr.tyBtnNo.bRtCompl	:= FALSE;
					tyP0204OpsMag3.tyMsgBoxSaveErr.tyBtnNo.bValue	:= FALSE;

					p_tyC0008MsgBox ACCESS ADR(tyP0204OpsMag3.tyMsgBoxHide);

					//Restore Param
					tyProdRcpCurrRcpWr	:= p_tyProdRcpCurrRcp2;

					tyP0204OpsMag3.tyParam.tyBtnSave.bRtCompl		:= FALSE;
					tyP0204OpsMag3.tyParam.tyBtnSave.bValue			:= FALSE;

					fUIInRtStatHide(ADR(tyP0204OpsMag3.tyParam.tyLyr.uiRtStat));

				END_IF

			END_IF

		ELSIF tyP0204OpsMag3.tyParam.tyBtnCancel.bRtCompl = TRUE THEN
			tyP0204OpsMag3.tyParam.tyBtnCancel.bRtCompl				:= FALSE;
			tyP0204OpsMag3.tyParam.tyBtnCancel.bValue				:= FALSE;

			fUIInRtStatHide(ADR(tyP0204OpsMag3.tyParam.tyLyr.uiRtStat));

		END_IF

	END_IF

	//Mask
	tyP0204OpsMag3.tyOps.tyBtnChgParam.uiMaskRtStat.0	:= p_tyUsrMgmtCurrAccessRgt.bChgParam AND p_bOpsStatusStop;

END_ACTION
```

#### Act_OptP0204InsertRmvMag.st
```iecst
ACTION Act_OptP0204InsertRmvMag:

	//Insert & Removed Magazine Manually Without Button Control
//	IF p_tyNtParamCurr.bProjBtnInsertRmvMag = FALSE THEN
//
//		IF p_bOpsStatusRun AND p_bOpsMagConvUL3InitDone THEN
//
//			fbMag3EntrySenOnTm(IN := p_tyDI.bMagConvEntSen3);
//
//			IF bNewMag3 = FALSE AND bRlsMag3 = FALSE THEN
//				IF p_bOpsMagConvUL3NewMagAllw AND fbMag3EntrySenOnTm.Q AND NOT p_bOpsMagConvUL3MagExitedWait THEN
//					bNewMag3	:= TRUE;
//				END_IF
//
//				IF p_bOpsMagConvUL3RlsMagAllw AND p_tyDI.bMagPresentSen3 AND p_tyDI.bOutShutterCloseRS AND p_tyBuffer3BffrStat.bBffrFull THEN
//					bRlsMag3	:= TRUE;
//				END_IF
//			END_IF
//
//			IF bNewMag3 = TRUE THEN
//
//				IF p_tyDI.bMag3FixedClampRS = TRUE AND p_tyDI.bMag3RemoteClampRS = TRUE THEN
//					bNewMag3	:= FALSE;
//				END_IF
//
//			ELSIF bRlsMag3 = TRUE THEN
//
//				IF p_tyDI.bMag3FixedUnclampRS = TRUE AND p_tyDI.bMag3RemoteUnclampRS = TRUE AND p_tyDI.bMagConvEntSen3 = TRUE THEN
//					bRlsMag3	:= FALSE;
//				END_IF
//
//			END_IF
//
//		ELSE
//
//			bNewMag3	:= FALSE;
//			bRlsMag3	:= FALSE;
//
//			fbMag3EntrySenOnTm(IN := FALSE);
//
//		END_IF
//
//	END_IF

END_ACTION
```

#### Act_OptP0204RstMnl.st
```iecst
ACTION Act_OptP0204RstMnl:

	IF eCurrPage <> UIP0204OpsMag3 AND eCurrPage <> UIP0003MMenu THEN
		bNewMag3	:= FALSE;
		bRlsMag3	:= FALSE;
		tyP0204OpsMag3.tyOps.tyBtnChgMag.bValue	:= FALSE;
		tyP0204OpsMag3.tyOps.tyBtnChgMag.bRtLk	:= FALSE;
		tyP0204OpsMag3.tyOps.tyBitmapChgMag.usiValueIdx	:= 0;

		tyP0003MMenu.tyMMenuBtn.tyBtnRlsNewMag3.bValue := FALSE;
		tyP0003MMenu.tyMMenuBtn.tyBtnRlsNewMag3.bRtLk  := FALSE;
		tyP0003MMenu.tyMMenuBtn.tyBtnRlsNewMag3.usiBitmapIdx := 0;
	END_IF

END_ACTION
```

#### Act_OptP0204AIVDat.st - not listed in the package file held
```iecst
ACTION Act_OptP0204AIVDat:

	//Show Change Mag Button only in Manual Exchane Mode
	tyP0204OpsMag3.tyOps.tyBtnChgMag.uiRtStat.0 := p_tyMcParamCurr.eMagExMode = McSetMagXcAutoMode AND p_tyMcParamCurr.eAGVComProtocol <> McSetAGVCommDisabled OR p_tyNtParamCurr.bProjLifterMagPlatform;
	tyP0204OpsMag3.tyOps.tyBitmapChgMag.uiRtStat.0 := p_tyMcParamCurr.eMagExMode = McSetMagXcAutoMode AND p_tyMcParamCurr.eAGVComProtocol <> McSetAGVCommDisabled OR p_tyNtParamCurr.bProjLifterMagPlatform;

	//LED Wifi
	tyP0204OpsMag3.tyOps.tyBtnAIVWifi.bValue	:= p_bAGVOnline;

	//Change Magazine
	IF p_tyNtParamCurr.bProjBtnInsertRmvMag = TRUE THEN

		IF EDGENEG(p_bOpsStatusRun) THEN
			bNewMag3	:= FALSE;
			tyP0204OpsMag3.tyOps.tyBtnChgMag.bRtLk	:= FALSE;
			tyP0204OpsMag3.tyOps.tyBtnChgMag.bRtCompl	:= FALSE;
			tyP0204OpsMag3.tyOps.tyBtnChgMag.bValue		:= FALSE;
		END_IF

		IF tyP0204OpsMag3.tyOps.tyBtnChgMag.bRtCompl = TRUE THEN
			tyP0204OpsMag3.tyOps.tyBtnChgMag.bRtCompl	:= FALSE;
			bNewMag3	:= p_bOpsMagConvUL3NewMagAllw;
			bRlsMag3	:= p_bOpsMagConvUL3RlsMagAllw;

		END_IF

		IF bNewMag3 = TRUE THEN
			tyP0204OpsMag3.tyOps.tyBitmapChgMag.usiValueIdx	:= 1;
			IF p_tyDI.bMag3FixedUnclampRS = FALSE THEN
				bNewMag3	:= FALSE;
				tyP0204OpsMag3.tyOps.tyBtnChgMag.bValue	:= FALSE;
				tyP0204OpsMag3.tyOps.tyBtnChgMag.bRtLk	:= FALSE;
				tyP0204OpsMag3.tyOps.tyBitmapChgMag.usiValueIdx	:= 0;
			END_IF

		ELSIF bRlsMag3 = TRUE THEN
			tyP0204OpsMag3.tyOps.tyBitmapChgMag.usiValueIdx	:= 1;
			IF p_tyNtParamCurr.eCustomerReq = Siemens THEN
				IF p_bOpsMagConvUL3EjectMESStep  THEN //FOR MES
					bRlsMag3	:= FALSE;
					tyP0204OpsMag3.tyOps.tyBtnChgMag.bValue	:= FALSE;
					tyP0204OpsMag3.tyOps.tyBtnChgMag.bRtLk	:= FALSE;
					tyP0204OpsMag3.tyOps.tyBitmapChgMag.usiValueIdx	:= 0;
				END_IF
			ELSIF (p_tyDI.bMag3FixedUnclampRS = TRUE AND p_tyDI.bMagPresentSen3 = FALSE) THEN
				bRlsMag3	:= FALSE;
				tyP0204OpsMag3.tyOps.tyBtnChgMag.bValue	:= FALSE;
				tyP0204OpsMag3.tyOps.tyBtnChgMag.bRtLk	:= FALSE;
				tyP0204OpsMag3.tyOps.tyBitmapChgMag.usiValueIdx	:= 0;
			END_IF

		ELSIF p_bAlarmErr THEN
			bNewMag3	:= FALSE;
			bRlsMag3	:= FALSE;
			tyP0204OpsMag3.tyOps.tyBtnChgMag.bValue	:= FALSE;
			tyP0204OpsMag3.tyOps.tyBtnChgMag.bRtLk	:= FALSE;
			tyP0204OpsMag3.tyOps.tyBitmapChgMag.usiValueIdx	:= 0;
		END_IF

		IF p_tyDI.bMagPresentSen3 AND p_tyDI.bMagConvEntSen3 = FALSE THEN
			tyP0204OpsMag3.tyOps.tyBtnChgMag.usiTxtIdx	:= 1;
		ELSE
			tyP0204OpsMag3.tyOps.tyBtnChgMag.usiTxtIdx	:= 0;
		END_IF

		IF (p_bOpsMagConvUL3NewMagAllw AND p_tyBuffer3BffrStat.bBffrMty)
			OR p_bOpsMagConvUL3RlsMagAllw
			OR p_bBufferMagRemoved3
			THEN //AND p_tyDI.bOutShutterCloseRS
			fUIInRtStatHide(ADR(tyP0204OpsMag3.tyOps.tyBtnChgMag.uiMaskRtStat));
		ELSE
			fUIInRtStatOff(ADR(tyP0204OpsMag3.tyOps.tyBtnChgMag.uiMaskRtStat));
		END_IF

	END_IF

END_ACTION
```

#### Act_EntP0205Disp.st
```iecst
ACTION Act_EntP0205Disp:

	//Access Address
	p_tyC0004Navi ACCESS ADR(tyP0205OpsAIV.tyNaviBack);

	p_tyC0005Main ACCESS ADR(tyCommon.tyMain);

	p_tyC0007Notif ACCESS ADR(tyCommon.tyNotif);

	p_tyC0008MsgBox ACCESS ADR(tyP0205OpsAIV.tyMsgBoxHide);

	p_tyC0009Info ACCESS ADR(tyCommon.tyInfo);

	p_tyP0205IOMonitor ACCESS ADR(tyP0205OpsAIV.tyIOMonitor);

	tyP0205OpsAIV.tyIOMonitor.tyBitmapAIVSLarge1.uiRtStat.0 := p_tyMcParamCurr.bAIVSizeDisabled OR p_tyMcParamCurr.eAGVComProtocol = McSetAGVTCPEnableTCP ;
	tyP0205OpsAIV.tyIOMonitor.tyBitmapAIVSLarge2.uiRtStat.0 := p_tyMcParamCurr.bAIVSizeDisabled OR p_tyMcParamCurr.eAGVComProtocol = McSetAGVTCPEnableTCP ;
	tyP0205OpsAIV.tyIOMonitor.tyBitmapAIVSLarge3.uiRtStat.0 := p_tyMcParamCurr.bAIVSizeDisabled OR p_tyMcParamCurr.eAGVComProtocol = McSetAGVTCPEnableTCP ;
	tyP0205OpsAIV.tyIOMonitor.tyBitmapAIVSLarge4.uiRtStat.0 := p_tyMcParamCurr.bAIVSizeDisabled OR p_tyMcParamCurr.eAGVComProtocol = McSetAGVTCPEnableTCP ;

	tyP0205OpsAIV.tyIOMonitor.tyBitmapMagSLarge1.uiRtStat.0 := p_tyMcParamCurr.bAIVSizeDisabled;
	tyP0205OpsAIV.tyIOMonitor.tyBitmapMagSLarge2.uiRtStat.0 := p_tyMcParamCurr.bAIVSizeDisabled;
	tyP0205OpsAIV.tyIOMonitor.tyBitmapMagSLarge3.uiRtStat.0 := p_tyMcParamCurr.bAIVSizeDisabled;
	tyP0205OpsAIV.tyIOMonitor.tyBitmapMagSLarge4.uiRtStat.0 := p_tyMcParamCurr.bAIVSizeDisabled;

	CASE p_tyMcParamCurr.eAGVComProtocol OF
		McSetAGVCommOPCUA:
			tyP0205OpsAIV.tyIOMonitor.tyTxtAIVCommProtocol.usiValueIdx := 0;

		McSetAGVCommHardIO:
			tyP0205OpsAIV.tyIOMonitor.tyTxtAIVCommProtocol.usiValueIdx := 1;

		McSetAGVCommDisabled:
			tyP0205OpsAIV.tyIOMonitor.tyTxtAIVCommProtocol.usiValueIdx := 2;

		McSetAGVTCPEnableTCP:
			tyP0205OpsAIV.tyIOMonitor.tyTxtAIVCommProtocol.uiRtStat := TRUE;
		McSetAGVTCPDisableTCP:
			tyP0205OpsAIV.tyIOMonitor.tyTxtAIVCommProtocol.uiRtStat := TRUE;
	END_CASE

END_ACTION
```

#### Act_OptP0205Navi.st
```iecst
ACTION Act_OptP0205Navi:

	IF tyP0205OpsAIV.tyNaviBack.tyBtnBack.bRtCompl = TRUE THEN
		tyP0205OpsAIV.tyNaviBack.tyBtnBack.bRtCompl	:= FALSE;
		tyP0205OpsAIV.tyNaviBack.tyBtnBack.bValue		:= FALSE;

		eChgPage	:= UIP0200OpsGen;

	ELSIF tyP0205OpsAIV.tyIOMonitor.tyHotspotClose.bRtCompl = TRUE THEN
		tyP0205OpsAIV.tyIOMonitor.tyHotspotClose.bRtCompl	:= FALSE;

		eChgPage	:= UIP0200OpsGen;

	END_IF

END_ACTION
```

#### Act_OptP0205IOMonitor.st
```iecst
ACTION Act_OptP0205IOMonitor:

	//Digital Input
	//AIV Err
	IF p_tyDI.bSOT1AIVError THEN
		tyP0205OpsAIV.tyIOMonitor.tyBitmapAIVErr1.usiValueIdx		:= 2;
	ELSE
		tyP0205OpsAIV.tyIOMonitor.tyBitmapAIVErr1.usiValueIdx		:= 0;
	END_IF

	IF p_tyDI.bSOT2AIVError THEN
		tyP0205OpsAIV.tyIOMonitor.tyBitmapAIVErr2.usiValueIdx		:= 2;
	ELSE
		tyP0205OpsAIV.tyIOMonitor.tyBitmapAIVErr2.usiValueIdx		:= 0;
	END_IF

	IF p_tyDI.bSOT3AIVError THEN
		tyP0205OpsAIV.tyIOMonitor.tyBitmapAIVErr3.usiValueIdx		:= 2;
	ELSE
		tyP0205OpsAIV.tyIOMonitor.tyBitmapAIVErr3.usiValueIdx		:= 0;
	END_IF

	IF p_tyDI.bSOT4AIVError THEN
		tyP0205OpsAIV.tyIOMonitor.tyBitmapAIVErr4.usiValueIdx		:= 2;
	ELSE
		tyP0205OpsAIV.tyIOMonitor.tyBitmapAIVErr4.usiValueIdx		:= 0;
	END_IF

	//AIV Ready

	IF p_tyDI.bSOT1AIVReady THEN
		tyP0205OpsAIV.tyIOMonitor.tyBitmapAIVRdy1.usiValueIdx		:= 1;
	ELSIF ADR(p_bTCPSvrUBA) = 0 THEN //Prevent Service mode
		tyP0205OpsAIV.tyIOMonitor.tyBitmapAIVRdy1.usiValueIdx		:= 0;
	ELSIF p_bTCPSvrUBA THEN
		tyP0205OpsAIV.tyIOMonitor.tyBitmapAIVRdy1.usiValueIdx		:= 1;
	ELSE
		tyP0205OpsAIV.tyIOMonitor.tyBitmapAIVRdy1.usiValueIdx		:= 0;
	END_IF

	IF p_tyDI.bSOT2AIVReady  THEN
		tyP0205OpsAIV.tyIOMonitor.tyBitmapAIVRdy2.usiValueIdx		:= 1;
	ELSIF ADR(p_bTCPSvrUBA2) = 0 THEN
		tyP0205OpsAIV.tyIOMonitor.tyBitmapAIVRdy2.usiValueIdx		:= 0;
	ELSIF p_bTCPSvrUBA2 THEN
		tyP0205OpsAIV.tyIOMonitor.tyBitmapAIVRdy2.usiValueIdx		:= 1;
	ELSE
		tyP0205OpsAIV.tyIOMonitor.tyBitmapAIVRdy2.usiValueIdx		:= 0;
	END_IF

	IF p_tyDI.bSOT3AIVReady THEN
		tyP0205OpsAIV.tyIOMonitor.tyBitmapAIVRdy3.usiValueIdx		:= 1;
	ELSE
		tyP0205OpsAIV.tyIOMonitor.tyBitmapAIVRdy3.usiValueIdx		:= 0;
	END_IF

	IF p_tyDI.bSOT4AIVReady THEN
		tyP0205OpsAIV.tyIOMonitor.tyBitmapAIVRdy4.usiValueIdx		:= 1;
	ELSE
		tyP0205OpsAIV.tyIOMonitor.tyBitmapAIVRdy4.usiValueIdx		:= 0;
	END_IF

	//AIV Available
	IF p_tyDI.bSOT1AIVAvailable  THEN
		tyP0205OpsAIV.tyIOMonitor.tyBitmapAIVAvail1.usiValueIdx		:= 1;
	ELSIF ADR(p_bTCPSvrDSB) = 0 THEN
		tyP0205OpsAIV.tyIOMonitor.tyBitmapAIVAvail1.usiValueIdx		:= 0;
	ELSIF p_bTCPSvrDSB THEN
		tyP0205OpsAIV.tyIOMonitor.tyBitmapAIVAvail1.usiValueIdx		:= 1;
	ELSE
		tyP0205OpsAIV.tyIOMonitor.tyBitmapAIVAvail1.usiValueIdx		:= 0;
	END_IF

	IF p_tyDI.bSOT2AIVAvailable  THEN
		tyP0205OpsAIV.tyIOMonitor.tyBitmapAIVAvail2.usiValueIdx		:= 1;
	ELSIF ADR(p_bTCPSvrDSB2) = 0 THEN
		tyP0205OpsAIV.tyIOMonitor.tyBitmapAIVAvail2.usiValueIdx		:= 0;
	ELSIF p_bTCPSvrDSB2 THEN
		tyP0205OpsAIV.tyIOMonitor.tyBitmapAIVAvail2.usiValueIdx		:= 1;
	ELSE
		tyP0205OpsAIV.tyIOMonitor.tyBitmapAIVAvail2.usiValueIdx		:= 0;
	END_IF

	IF p_tyDI.bSOT3AIVAvailable THEN
		tyP0205OpsAIV.tyIOMonitor.tyBitmapAIVAvail3.usiValueIdx		:= 1;
	ELSE
		tyP0205OpsAIV.tyIOMonitor.tyBitmapAIVAvail3.usiValueIdx		:= 0;
	END_IF

	IF p_tyDI.bSOT4AIVAvailable THEN
		tyP0205OpsAIV.tyIOMonitor.tyBitmapAIVAvail4.usiValueIdx		:= 1;
	ELSE
		tyP0205OpsAIV.tyIOMonitor.tyBitmapAIVAvail4.usiValueIdx		:= 0;
	END_IF

	//AIV Size
	IF p_tyDI.bSOT1AIVSizeLarge THEN
		tyP0205OpsAIV.tyIOMonitor.tyBitmapAIVSLarge1.usiValueIdx		:= 1;
	ELSE
		tyP0205OpsAIV.tyIOMonitor.tyBitmapAIVSLarge1.usiValueIdx		:= 0;
	END_IF

	IF p_tyDI.bSOT2AIVSizeLarge THEN
		tyP0205OpsAIV.tyIOMonitor.tyBitmapAIVSLarge2.usiValueIdx		:= 1;
	ELSE
		tyP0205OpsAIV.tyIOMonitor.tyBitmapAIVSLarge2.usiValueIdx		:= 0;
	END_IF

	IF p_tyDI.bSOT3AIVSizeLarge THEN
		tyP0205OpsAIV.tyIOMonitor.tyBitmapAIVSLarge3.usiValueIdx		:= 1;
	ELSE
		tyP0205OpsAIV.tyIOMonitor.tyBitmapAIVSLarge3.usiValueIdx		:= 0;
	END_IF

	IF p_tyDI.bSOT4AIVSizeLarge THEN
		tyP0205OpsAIV.tyIOMonitor.tyBitmapAIVSLarge4.usiValueIdx		:= 1;
	ELSE
		tyP0205OpsAIV.tyIOMonitor.tyBitmapAIVSLarge4.usiValueIdx		:= 0;
	END_IF

	tyP0205OpsAIV.tyIOMonitor.tyBtnAIVSotRCVOk1.bValue			:= p_tyDI.bSOT1Receive;
	tyP0205OpsAIV.tyIOMonitor.tyBtnAIVSotRCVOk2.bValue			:= p_tyDI.bSOT2Receive;
	tyP0205OpsAIV.tyIOMonitor.tyBtnAIVSotRCVOk3.bValue			:= p_tyDI.bSOT3Receive;
	tyP0205OpsAIV.tyIOMonitor.tyBtnAIVSotRCVOk4.bValue			:= p_tyDI.bSOT4Receive;

	//Digital Output
	//Mag Error
	IF p_tyDO.bSOT1MagError THEN
		tyP0205OpsAIV.tyIOMonitor.tyBitmapMagErr1.usiValueIdx		:= 2;
	ELSE
		tyP0205OpsAIV.tyIOMonitor.tyBitmapMagErr1.usiValueIdx		:= 0;
	END_IF

	IF p_tyDO.bSOT2MagError THEN
		tyP0205OpsAIV.tyIOMonitor.tyBitmapMagErr2.usiValueIdx		:= 2;
	ELSE
		tyP0205OpsAIV.tyIOMonitor.tyBitmapMagErr2.usiValueIdx		:= 0;
	END_IF

	IF p_tyDO.bSOT3MagError THEN
		tyP0205OpsAIV.tyIOMonitor.tyBitmapMagErr3.usiValueIdx		:= 2;
	ELSE
		tyP0205OpsAIV.tyIOMonitor.tyBitmapMagErr3.usiValueIdx		:= 0;
	END_IF

	IF p_tyDO.bSOT4MagError THEN
		tyP0205OpsAIV.tyIOMonitor.tyBitmapMagErr4.usiValueIdx		:= 2;
	ELSE
		tyP0205OpsAIV.tyIOMonitor.tyBitmapMagErr4.usiValueIdx		:= 0;
	END_IF

	//Mag Ready
	IF p_tyDO.bSOT1MagReady THEN
		tyP0205OpsAIV.tyIOMonitor.tyBitmapMagRdy1.usiValueIdx		:= 1;
	ELSE
		tyP0205OpsAIV.tyIOMonitor.tyBitmapMagRdy1.usiValueIdx		:= 0;
	END_IF

	IF p_tyDO.bSOT2MagReady THEN
		tyP0205OpsAIV.tyIOMonitor.tyBitmapMagRdy2.usiValueIdx		:= 1;
	ELSE
		tyP0205OpsAIV.tyIOMonitor.tyBitmapMagRdy2.usiValueIdx		:= 0;
	END_IF

	IF p_tyDO.bSOT3MagReady THEN
		tyP0205OpsAIV.tyIOMonitor.tyBitmapMagRdy3.usiValueIdx		:= 1;
	ELSE
		tyP0205OpsAIV.tyIOMonitor.tyBitmapMagRdy3.usiValueIdx		:= 0;
	END_IF

	IF p_tyDO.bSOT4MagReady THEN
		tyP0205OpsAIV.tyIOMonitor.tyBitmapMagRdy4.usiValueIdx		:= 1;
	ELSE
		tyP0205OpsAIV.tyIOMonitor.tyBitmapMagRdy4.usiValueIdx		:= 0;
	END_IF

	//Mag Available
	IF p_tyDO.bSOT1MagAvailable THEN
		tyP0205OpsAIV.tyIOMonitor.tyBitmapMagAvail1.usiValueIdx		:= 1;
	ELSE
		tyP0205OpsAIV.tyIOMonitor.tyBitmapMagAvail1.usiValueIdx		:= 0;
	END_IF

	IF p_tyDO.bSOT2MagAvailable THEN
		tyP0205OpsAIV.tyIOMonitor.tyBitmapMagAvail2.usiValueIdx		:= 1;
	ELSE
		tyP0205OpsAIV.tyIOMonitor.tyBitmapMagAvail2.usiValueIdx		:= 0;
	END_IF

	IF p_tyDO.bSOT3MagAvailable THEN
		tyP0205OpsAIV.tyIOMonitor.tyBitmapMagAvail3.usiValueIdx		:= 1;
	ELSE
		tyP0205OpsAIV.tyIOMonitor.tyBitmapMagAvail3.usiValueIdx		:= 0;
	END_IF

	IF p_tyDO.bSOT4MagAvailable THEN
		tyP0205OpsAIV.tyIOMonitor.tyBitmapMagAvail4.usiValueIdx		:= 1;
	ELSE
		tyP0205OpsAIV.tyIOMonitor.tyBitmapMagAvail4.usiValueIdx		:= 0;
	END_IF

	//Mag Size
	IF p_tyDO.bSOT1MagSizeLarge THEN
		tyP0205OpsAIV.tyIOMonitor.tyBitmapMagSLarge1.usiValueIdx		:= 1;
	ELSE
		tyP0205OpsAIV.tyIOMonitor.tyBitmapMagSLarge1.usiValueIdx		:= 0;
	END_IF

	IF p_tyDO.bSOT2MagSizeLarge THEN
		tyP0205OpsAIV.tyIOMonitor.tyBitmapMagSLarge2.usiValueIdx		:= 1;
	ELSE
		tyP0205OpsAIV.tyIOMonitor.tyBitmapMagSLarge2.usiValueIdx		:= 0;
	END_IF

	IF p_tyDO.bSOT3MagSizeLarge THEN
		tyP0205OpsAIV.tyIOMonitor.tyBitmapMagSLarge3.usiValueIdx		:= 1;
	ELSE
		tyP0205OpsAIV.tyIOMonitor.tyBitmapMagSLarge3.usiValueIdx		:= 0;
	END_IF

	IF p_tyDO.bSOT4MagSizeLarge THEN
		tyP0205OpsAIV.tyIOMonitor.tyBitmapMagSLarge4.usiValueIdx		:= 1;
	ELSE
		tyP0205OpsAIV.tyIOMonitor.tyBitmapMagSLarge4.usiValueIdx		:= 0;
	END_IF

	//MES Name
	tyP0205OpsAIV.tyIOMonitor.tyStringMesName.sValue			:= p_tyTagFromMes.sMESName;

	CASE p_tyMcParamCurr.eAGVComProtocol OF
		McSetAGVCommOPCUA:
			//Req To Bring
			tyP0205OpsAIV.tyIOMonitor.tyBtnReqAIVToBring1.bValue		:= p_tyTagToMes.tyTagStatOfPlatforms[1].bReqAIVToBring;
			tyP0205OpsAIV.tyIOMonitor.tyBtnReqAIVToBring2.bValue		:= p_tyTagToMes.tyTagStatOfPlatforms[2].bReqAIVToBring;
			tyP0205OpsAIV.tyIOMonitor.tyBtnReqAIVToBring3.bValue		:= p_tyTagToMes.tyTagStatOfPlatforms[3].bReqAIVToBring;
			tyP0205OpsAIV.tyIOMonitor.tyBtnReqAIVToBring4.bValue		:= p_tyTagToMes.tyTagStatOfPlatforms[4].bReqAIVToBring;
			//Req To Get
			tyP0205OpsAIV.tyIOMonitor.tyBtnReqAIVToGet1.bValue		:= p_tyTagToMes.tyTagStatOfPlatforms[1].bReqAIVToGet;
			tyP0205OpsAIV.tyIOMonitor.tyBtnReqAIVToGet2.bValue		:= p_tyTagToMes.tyTagStatOfPlatforms[2].bReqAIVToGet;
			tyP0205OpsAIV.tyIOMonitor.tyBtnReqAIVToGet3.bValue		:= p_tyTagToMes.tyTagStatOfPlatforms[3].bReqAIVToGet;
			tyP0205OpsAIV.tyIOMonitor.tyBtnReqAIVToGet4.bValue		:= p_tyTagToMes.tyTagStatOfPlatforms[4].bReqAIVToGet;

			tyP0205OpsAIV.tyIOMonitor.tyBtnMESActive.bValue				:= p_tyTagFromMes.bActive;
		McSetAGVCommHardIO:
			//Req To Bring
			tyP0205OpsAIV.tyIOMonitor.tyBtnReqAIVToBring1.bValue		:= p_tyDO.bMag1ReqToBring;
			tyP0205OpsAIV.tyIOMonitor.tyBtnReqAIVToBring2.bValue		:= p_tyDO.bMag2ReqToBring;
			tyP0205OpsAIV.tyIOMonitor.tyBtnReqAIVToBring3.bValue		:= p_tyDO.bMag3ReqToBring;
			tyP0205OpsAIV.tyIOMonitor.tyBtnReqAIVToBring4.bValue		:= p_tyDO.bMag4ReqToBring;
			//Req To Get
			tyP0205OpsAIV.tyIOMonitor.tyBtnReqAIVToGet1.bValue		:= p_tyDO.bMag1ReqToGet;
			tyP0205OpsAIV.tyIOMonitor.tyBtnReqAIVToGet2.bValue		:= p_tyDO.bMag2ReqToGet;
			tyP0205OpsAIV.tyIOMonitor.tyBtnReqAIVToGet3.bValue		:= p_tyDO.bMag3ReqToGet;
			tyP0205OpsAIV.tyIOMonitor.tyBtnReqAIVToGet4.bValue		:= p_tyDO.bMag4ReqToGet;

			tyP0205OpsAIV.tyIOMonitor.tyBtnMESActive.bValue				:= p_tyDI.bFleetManagerReady;
		McSetAGVCommDisabled:
			//Req To Bring
			tyP0205OpsAIV.tyIOMonitor.tyBtnReqAIVToBring1.bValue		:= FALSE;
			tyP0205OpsAIV.tyIOMonitor.tyBtnReqAIVToBring2.bValue		:= FALSE;
			tyP0205OpsAIV.tyIOMonitor.tyBtnReqAIVToBring3.bValue		:= FALSE;
			tyP0205OpsAIV.tyIOMonitor.tyBtnReqAIVToBring4.bValue		:= FALSE;
			//Req To Get
			tyP0205OpsAIV.tyIOMonitor.tyBtnReqAIVToGet1.bValue		:= FALSE;
			tyP0205OpsAIV.tyIOMonitor.tyBtnReqAIVToGet2.bValue		:= FALSE;
			tyP0205OpsAIV.tyIOMonitor.tyBtnReqAIVToGet3.bValue		:= FALSE;
			tyP0205OpsAIV.tyIOMonitor.tyBtnReqAIVToGet4.bValue		:= FALSE;

			tyP0205OpsAIV.tyIOMonitor.tyBtnMESActive.bValue	:= FALSE;
	END_CASE

END_ACTION
```

#### Act_OptP0205RstMnl.st
```iecst
ACTION Act_OptP0205RstMnl:

END_ACTION
```

#### Act_EntP0206Disp.st
```iecst
ACTION Act_EntP0206Disp:

	//Access Address
	p_tyC0004Navi ACCESS ADR(tyP0206OpsMagConv1.tyNaviBack);

	p_tyC0005Main ACCESS ADR(tyCommon.tyMain);

	p_tyC0007Notif ACCESS ADR(tyCommon.tyNotif);

	p_tyC0008MsgBox ACCESS ADR(tyP0206OpsMagConv1.tyMsgBoxHide);

	p_tyC0009Info ACCESS ADR(tyCommon.tyInfo);

	p_tyC0011RcpPopUp ACCESS ADR(tyP0206OpsMagConv1.tyRcpPopUp);

	p_tyP0206OpsMagConv1 ACCESS ADR(tyP0206OpsMagConv1.tyOps);
	p_tyP0206MagConvIOMonitor1 ACCESS ADR(tyP0206OpsMagConv1.tyIOMonitor);
	p_tyP0206MagConvBypsInitConv1 ACCESS ADR(tyP0206OpsMagConv1.tyBypsInitConv);

	//Display
	fUIInRtStatHide(ADR(tyP0206OpsMagConv1.tyIOMonitor.tyLyr.uiRtStat));

	tyP0206OpsMagConv1.tyOps.tyBtnChgParam.uiRtStat.0	:= NOT(p_tyMcParamCurr.bChgParamEn);

END_ACTION
```

#### Act_OptP0206Navi.st
```iecst
ACTION Act_OptP0206Navi:

	IF tyP0206OpsMagConv1.tyNaviBack.tyBtnBack.bRtCompl = TRUE THEN
		tyP0206OpsMagConv1.tyNaviBack.tyBtnBack.bRtCompl	:= FALSE;
		tyP0206OpsMagConv1.tyNaviBack.tyBtnBack.bValue	:= FALSE;

		eChgPage	:= UIP0200OpsGen;

	END_IF

END_ACTION
```

#### Act_OptP0206UpdtDat.st
```iecst
ACTION Act_OptP0206UpdtDat:

	//Status
	fbMcStatUpdtTm(IN := TRUE);
	IF fbMcStatUpdtTm.Q = TRUE THEN
		fbMcStatUpdtTm(IN := FALSE);

		tyP0206OpsMagConv1.tyOps.tyStringMcTopStat.sValue	:= p_sOpsInMagConvStepTxt;
		tyP0206OpsMagConv1.tyOps.tyStringMcBtmStat.sValue	:= p_sOpsOutMagConvStepTxt;
	END_IF

	//Mode
	tyP0206OpsMagConv1.tyOps.tyTxtMod.usiValueIdx	:= p_tyProdRcpCurrRcp1.usiMcMod;

	//Width
	IF p_tyNtParamCurr.bAWPrep = TRUE AND p_tyMcParamCurr.bAWDis = FALSE THEN
		tyP0206OpsMagConv1.tyOps.tyNumWidth.diValue		:= p_tyMcParamCurr.diWidthAtHmPosInUM - p_diAWOpenActualPos;
		tyP0206OpsMagConv1.tyOps.tyNumWidth2.diValue	:= p_tyMcParamCurr.diWidthAtHmPosInUM - p_diAWOpenActualPos;
	ELSE
		tyP0206OpsMagConv1.tyOps.tyNumWidth.diValue		:= p_tyProdRcpCurrRcp1.diWidthInUM;
		tyP0206OpsMagConv1.tyOps.tyNumWidth2.diValue		:= p_tyProdRcpCurrRcp1.diWidthInUM2;
	END_IF

	//Program Info
	tyP0206OpsMagConv1.tyOps.tyStringProdNm.sValue		:= p_tyProdRcpCurrRcp1.sRcpNm;
	tyP0206OpsMagConv1.tyOps.tyNumMinSltRange.diValue		:= p_tyProdRcpCurrRcp1.diMinSltValue;
	tyP0206OpsMagConv1.tyOps.tyNumMaxSltRange.diValue		:= p_tyProdRcpCurrRcp1.diMaxSltValue;
	tyP0206OpsMagConv1.tyOps.tyBtnToptoBtm.bValue			:= p_tyProdRcpCurrRcp1.bTopToBtm;
	tyP0206OpsMagConv1.tyOps.tyNumPitch.diValue			:= p_tyProdRcpCurrRcp1.diPitch;

	//PCB Status
	IF p_bPshrConvHvBrd = TRUE THEN
		IF p_bPshrConvGdBrd = TRUE THEN
			tyP0206OpsMagConv1.tyOps.tyBitmapPCB.usiValueIdx	:= 1;
		ELSE
			tyP0206OpsMagConv1.tyOps.tyBitmapPCB.usiValueIdx	:= 2;
		END_IF
	ELSE
		tyP0206OpsMagConv1.tyOps.tyBitmapPCB.usiValueIdx	:= 0;
	END_IF

	//AIV TCP Bitmap
	IF p_tyNtParamCurr.bProjAGVPrep THEN
		tyP0206OpsMagConv1.tyOps.tyBtnAIVWifi.usiBitmapIdx := BOOL_TO_USINT (p_bTCPConnected);
	END_IF

	//Product Recipe 254
	tyP0206OpsMagConv1.tyOps.tyHotspotShowLRcp.uiRtStat.0 := NOT(tyP0206OpsMagConv1.tyOps.tyStringProdNm.sValue <> '');

	IF tyP0206OpsMagConv1.tyOps.tyHotspotShowLRcp.bRtCompl = TRUE THEN
		tyP0206OpsMagConv1.tyOps.tyHotspotShowLRcp.bRtCompl := FALSE;

		fUIInRtStatOff(ADR(tyP0206OpsMagConv1.tyRcpPopUp.tyLyr.uiRtStat));

		tyP0206OpsMagConv1.tyRcpPopUp.tyStringInfo.sValue  := p_tyProdRcpCurrRcp1.sRcpNm;

	ELSIF tyP0206OpsMagConv1.tyRcpPopUp.tyHotspotClose.bRtCompl = TRUE THEN
		tyP0206OpsMagConv1.tyRcpPopUp.tyHotspotClose.bRtCompl := FALSE;

		fUIInRtStatHide(ADR(tyP0206OpsMagConv1.tyRcpPopUp.tyLyr.uiRtStat));
	END_IF

END_ACTION
```

#### Act_OptP0206IOMonitor.st
```iecst
ACTION Act_OptP0206IOMonitor:

	IF tyP0206OpsMagConv1.tyOps.tyHotspotIOMonitor.bRtCompl = TRUE THEN
		tyP0206OpsMagConv1.tyOps.tyHotspotIOMonitor.bRtCompl	:= FALSE;

		fUIInRtStatOff(ADR(tyP0206OpsMagConv1.tyIOMonitor.tyLyr.uiRtStat));

		p_tyC0004Navi ACCESS ADR(tyP0206OpsMagConv1.tyNaviHide);

	ELSIF tyP0206OpsMagConv1.tyIOMonitor.tyHotspotClose.bRtCompl = TRUE THEN
		tyP0206OpsMagConv1.tyIOMonitor.tyHotspotClose.bRtCompl	:= FALSE;

		fUIInRtStatHide(ADR(tyP0206OpsMagConv1.tyIOMonitor.tyLyr.uiRtStat));

		p_tyC0004Navi ACCESS ADR(tyP0206OpsMagConv1.tyNaviBack);

	END_IF

	IF tyP0206OpsMagConv1.tyIOMonitor.tyLyr.uiRtStat.0 = FALSE THEN

		//Digital Input
		tyP0206OpsMagConv1.tyIOMonitor.tyBtnSafetyRlySig.bValue			:= p_tyDI.bSafetyRlySig;
		tyP0206OpsMagConv1.tyIOMonitor.tyBtnEStop.bValue				:= p_tyDI.bEStopSig;
		tyP0206OpsMagConv1.tyIOMonitor.tyBtnCoverSWSig.bValue			:= p_tyDI.bCoverSWSig;
		tyP0206OpsMagConv1.tyIOMonitor.tyBtnTopEntSen.bValue			:= p_tyDI.bInMagConvEntSen;
		tyP0206OpsMagConv1.tyIOMonitor.tyBtnTopMidSen.bValue			:= p_tyDI.bInMagConvMidSen;
		tyP0206OpsMagConv1.tyIOMonitor.tyBtnTopExtSen.bValue			:= p_tyDI.bInMagConvExtSen;
		tyP0206OpsMagConv1.tyIOMonitor.tyBtnBtmEntSen.bValue			:= p_tyDI.bOutMagConvEntSen;
		tyP0206OpsMagConv1.tyIOMonitor.tyBtnBtmMidSen.bValue			:= p_tyDI.bOutMagConvMidSen;
		tyP0206OpsMagConv1.tyIOMonitor.tyBtnBtmExtSen.bValue			:= p_tyDI.bOutMagConvExtSen;

		//Digital Output
		tyP0206OpsMagConv1.tyIOMonitor.tyBtnSafetyRlyRst.bValue			:= p_tyDO.bSafetyRlyRst;
		tyP0206OpsMagConv1.tyIOMonitor.tyBtnTLGreen.bValue				:= p_tyDO.bTLGreen;
		tyP0206OpsMagConv1.tyIOMonitor.tyBtnTLAmber.bValue				:= p_tyDO.bTLAmber;
		tyP0206OpsMagConv1.tyIOMonitor.tyBtnTLRed.bValue				:= p_tyDO.bTLRed;
		tyP0206OpsMagConv1.tyIOMonitor.tyBtnBuzzer.bValue				:= p_tyDO.bBuzzer;
		tyP0206OpsMagConv1.tyIOMonitor.tyBtnEntStprRet.bValue			:= p_tyDO.bEntTopStprUnblkCtrl;
		tyP0206OpsMagConv1.tyIOMonitor.tyBtnMidStprExt.bValue			:= p_tyDO.bMidTopStprUnblkCtrl;
		tyP0206OpsMagConv1.tyIOMonitor.tyBtnExtStprRet.bValue			:= p_tyDO.bExtTopStprUnblkCtrl;
		tyP0206OpsMagConv1.tyIOMonitor.tyBtnMidStprExt1.bValue			:= p_tyDO.bMidBtmStprUnblkCtrl;
		tyP0206OpsMagConv1.tyIOMonitor.tyBtnExtStprRet1.bValue			:= p_tyDO.bExtBtmStprUnblkCtrl;

	END_IF

END_ACTION
```

#### Act_EntP0207Disp.st
```iecst
ACTION Act_EntP0207Disp:

	//Access Address
	p_tyC0004Navi ACCESS ADR(tyP0207OpsMagConv2.tyNaviBack);

	p_tyC0005Main ACCESS ADR(tyCommon.tyMain);

	p_tyC0007Notif ACCESS ADR(tyCommon.tyNotif);

	p_tyC0008MsgBox ACCESS ADR(tyP0207OpsMagConv2.tyMsgBoxHide);

	p_tyC0009Info ACCESS ADR(tyCommon.tyInfo);

	p_tyC0011RcpPopUp ACCESS ADR(tyP0207OpsMagConv2.tyRcpPopUp);

	p_tyP0207OpsMagConv2 ACCESS ADR(tyP0207OpsMagConv2.tyOps);
	p_tyP0207MagConvIOMonitor2 ACCESS ADR(tyP0207OpsMagConv2.tyIOMonitor);
	p_tyP0207MagConvBypsInitConv2 ACCESS ADR(tyP0207OpsMagConv2.tyBypsInitConv);

	//Display
	fUIInRtStatHide(ADR(tyP0207OpsMagConv2.tyIOMonitor.tyLyr.uiRtStat));

	tyP0207OpsMagConv2.tyOps.tyBtnChgParam.uiRtStat.0	:= NOT(p_tyMcParamCurr.bChgParamEn);

END_ACTION
```

#### Act_OptP0207Navi.st
```iecst
ACTION Act_OptP0207Navi:

	IF tyP0207OpsMagConv2.tyNaviBack.tyBtnBack.bRtCompl = TRUE THEN
		tyP0207OpsMagConv2.tyNaviBack.tyBtnBack.bRtCompl	:= FALSE;
		tyP0207OpsMagConv2.tyNaviBack.tyBtnBack.bValue	:= FALSE;

		eChgPage	:= UIP0200OpsGen;

	END_IF

END_ACTION
```

#### Act_OptP0207UpdtDat.st
```iecst
ACTION Act_OptP0207UpdtDat:

	//Status
	fbMcStatUpdtTm(IN := TRUE);
	IF fbMcStatUpdtTm.Q = TRUE THEN
		fbMcStatUpdtTm(IN := FALSE);

		tyP0207OpsMagConv2.tyOps.tyStringMcTopStat.sValue	:= p_sOpsInMagConvStepTxt1;
		tyP0207OpsMagConv2.tyOps.tyStringMcBtmStat.sValue	:= p_sOpsOutMagConvStepTxt1;
	END_IF

	//Mode
	tyP0207OpsMagConv2.tyOps.tyTxtMod.usiValueIdx	:= p_tyProdRcpCurrRcp1.usiMcMod;

	//Width
	IF p_tyNtParamCurr.bAWPrep = TRUE AND p_tyMcParamCurr.bAWDis = FALSE THEN
		tyP0207OpsMagConv2.tyOps.tyNumWidth.diValue		:= p_tyMcParamCurr.diWidthAtHmPosInUM - p_diAWOpenActualPos;
		tyP0207OpsMagConv2.tyOps.tyNumWidth2.diValue	:= p_tyMcParamCurr.diWidthAtHmPosInUM - p_diAWOpenActualPos;
	ELSE
		tyP0207OpsMagConv2.tyOps.tyNumWidth.diValue		:= p_tyProdRcpCurrRcp1.diWidthInUM;
		tyP0207OpsMagConv2.tyOps.tyNumWidth2.diValue		:= p_tyProdRcpCurrRcp1.diWidthInUM2;
	END_IF

	//Program Info
	tyP0207OpsMagConv2.tyOps.tyStringProdNm.sValue		:= p_tyProdRcpCurrRcp1.sRcpNm;
	tyP0207OpsMagConv2.tyOps.tyNumMinSltRange.diValue		:= p_tyProdRcpCurrRcp1.diMinSltValue;
	tyP0207OpsMagConv2.tyOps.tyNumMaxSltRange.diValue		:= p_tyProdRcpCurrRcp1.diMaxSltValue;
	tyP0207OpsMagConv2.tyOps.tyBtnToptoBtm.bValue			:= p_tyProdRcpCurrRcp1.bTopToBtm;
	tyP0207OpsMagConv2.tyOps.tyNumPitch.diValue			:= p_tyProdRcpCurrRcp1.diPitch;

	//PCB Status
	IF p_bPshrConvHvBrd = TRUE THEN
		IF p_bPshrConvGdBrd = TRUE THEN
			tyP0207OpsMagConv2.tyOps.tyBitmapPCB.usiValueIdx	:= 1;
		ELSE
			tyP0207OpsMagConv2.tyOps.tyBitmapPCB.usiValueIdx	:= 2;
		END_IF
	ELSE
		tyP0207OpsMagConv2.tyOps.tyBitmapPCB.usiValueIdx	:= 0;
	END_IF

	//AIV TCP Bitmap
	IF p_tyNtParamCurr.bProjAGVPrep THEN
		tyP0207OpsMagConv2.tyOps.tyBtnAIVWifi.usiBitmapIdx := BOOL_TO_USINT (p_bTCPConnected);
	END_IF
	//Product Recipe 254
	tyP0207OpsMagConv2.tyOps.tyHotspotShowLRcp.uiRtStat.0 := NOT(tyP0207OpsMagConv2.tyOps.tyStringProdNm.sValue <> '');

	IF tyP0207OpsMagConv2.tyOps.tyHotspotShowLRcp.bRtCompl = TRUE THEN
		tyP0207OpsMagConv2.tyOps.tyHotspotShowLRcp.bRtCompl := FALSE;

		fUIInRtStatOff(ADR(tyP0207OpsMagConv2.tyRcpPopUp.tyLyr.uiRtStat));

		tyP0207OpsMagConv2.tyRcpPopUp.tyStringInfo.sValue  := p_tyProdRcpCurrRcp1.sRcpNm;

	ELSIF tyP0207OpsMagConv2.tyRcpPopUp.tyHotspotClose.bRtCompl = TRUE THEN
		tyP0207OpsMagConv2.tyRcpPopUp.tyHotspotClose.bRtCompl := FALSE;

		fUIInRtStatHide(ADR(tyP0207OpsMagConv2.tyRcpPopUp.tyLyr.uiRtStat));
	END_IF

END_ACTION
```

#### Act_OptP0207IOMonitor.st
```iecst
ACTION Act_OptP0207IOMonitor:

	IF tyP0207OpsMagConv2.tyOps.tyHotspotIOMonitor.bRtCompl = TRUE THEN
		tyP0207OpsMagConv2.tyOps.tyHotspotIOMonitor.bRtCompl	:= FALSE;

		fUIInRtStatOff(ADR(tyP0207OpsMagConv2.tyIOMonitor.tyLyr.uiRtStat));

		p_tyC0004Navi ACCESS ADR(tyP0207OpsMagConv2.tyNaviHide);

	ELSIF tyP0207OpsMagConv2.tyIOMonitor.tyHotspotClose.bRtCompl = TRUE THEN
		tyP0207OpsMagConv2.tyIOMonitor.tyHotspotClose.bRtCompl	:= FALSE;

		fUIInRtStatHide(ADR(tyP0207OpsMagConv2.tyIOMonitor.tyLyr.uiRtStat));

		p_tyC0004Navi ACCESS ADR(tyP0207OpsMagConv2.tyNaviBack);

	END_IF

	IF tyP0207OpsMagConv2.tyIOMonitor.tyLyr.uiRtStat.0 = FALSE THEN

		//Digital Input
		tyP0207OpsMagConv2.tyIOMonitor.tyBtnSafetyRlySig.bValue			:= p_tyDI.bSafetyRlySig;
		tyP0207OpsMagConv2.tyIOMonitor.tyBtnEStop.bValue				:= p_tyDI.bEStopSig;
		tyP0207OpsMagConv2.tyIOMonitor.tyBtnCoverSWSig.bValue			:= p_tyDI.bCoverSWSig;
		tyP0207OpsMagConv2.tyIOMonitor.tyBtnTopEntSen.bValue			:= p_tyDI.bInMagConv2EntSen;
		tyP0207OpsMagConv2.tyIOMonitor.tyBtnTopMidSen.bValue			:= p_tyDI.bInMagConv2MidSen;
		tyP0207OpsMagConv2.tyIOMonitor.tyBtnTopExtSen.bValue			:= p_tyDI.bInMagConv2ExtSen;
		tyP0207OpsMagConv2.tyIOMonitor.tyBtnBtmEntSen.bValue			:= p_tyDI.bOutMagConv2EntSen;
		tyP0207OpsMagConv2.tyIOMonitor.tyBtnBtmMidSen.bValue			:= p_tyDI.bOutMagConv2MidSen;
		tyP0207OpsMagConv2.tyIOMonitor.tyBtnBtmExtSen.bValue			:= p_tyDI.bOutMagConv2ExtSen;

		//Digital Output
		tyP0207OpsMagConv2.tyIOMonitor.tyBtnSafetyRlyRst.bValue			:= p_tyDO.bSafetyRlyRst;
		tyP0207OpsMagConv2.tyIOMonitor.tyBtnTLGreen.bValue				:= p_tyDO.bTLGreen;
		tyP0207OpsMagConv2.tyIOMonitor.tyBtnTLAmber.bValue				:= p_tyDO.bTLAmber;
		tyP0207OpsMagConv2.tyIOMonitor.tyBtnTLRed.bValue				:= p_tyDO.bTLRed;
		tyP0207OpsMagConv2.tyIOMonitor.tyBtnBuzzer.bValue				:= p_tyDO.bBuzzer;
		tyP0207OpsMagConv2.tyIOMonitor.tyBtnEntStprRet.bValue			:= p_tyDO.bEntTopStprUnblkCtrl2;
		tyP0207OpsMagConv2.tyIOMonitor.tyBtnMidStprExt.bValue			:= p_tyDO.bMidTopStprUnblkCtrl2;
		tyP0207OpsMagConv2.tyIOMonitor.tyBtnExtStprRet.bValue			:= p_tyDO.bExtTopStprUnblkCtrl2;
		tyP0207OpsMagConv2.tyIOMonitor.tyBtnMidStprExt1.bValue			:= p_tyDO.bMidBtmStprUnblkCtrl2;
		tyP0207OpsMagConv2.tyIOMonitor.tyBtnExtStprRet1.bValue			:= p_tyDO.bExtBtmStprUnblkCtrl2;

	END_IF

END_ACTION
```

#### Act_OptP0200ToP0204_P0003AccDat.st
```iecst
ACTION Act_OptP0200ToP0204_P0003AccDat:

//	IF EDGENEG(p_bLFFollowerProdAccDataMnl OR p_bLCSLFAccDataMnl OR p_bUSHermesAAccDataMnl OR p_bUSHermesBAccDataMnl) THEN
//		bProdAccData	:= FALSE;
//	END_IF

	//Control
	IF (tyP0200OpsGen.tyOps.tyBtnAccDat.bRtCompl = TRUE)		OR (tyP0201OpsTravLifter.tyOps.tyBtnAccDat.bRtCompl = TRUE)
		OR (tyP0202OpsMag1.tyOps.tyBtnAccDat.bRtCompl = TRUE)	OR (tyP0203OpsMag2.tyOps.tyBtnAccDat.bRtCompl = TRUE)
		OR (tyP0204OpsMag3.tyOps.tyBtnAccDat.bRtCompl = TRUE) 	OR (tyP0206OpsMagConv1.tyOps.tyBtnAccDat.bRtCompl = TRUE)
		OR (tyP0207OpsMagConv2.tyOps.tyBtnAccDat.bRtCompl = TRUE) OR tyP0003MMenu.tyMMenuBtn.tyBtnAccDat.bRtCompl THEN

		tyP0200OpsGen.tyOps.tyBtnAccDat.bRtCompl		:= FALSE;
		tyP0201OpsTravLifter.tyOps.tyBtnAccDat.bRtCompl	:= FALSE;
		tyP0202OpsMag1.tyOps.tyBtnAccDat.bRtCompl		:= FALSE;
		tyP0203OpsMag2.tyOps.tyBtnAccDat.bRtCompl		:= FALSE;
		tyP0204OpsMag3.tyOps.tyBtnAccDat.bRtCompl		:= FALSE;
		tyP0206OpsMagConv1.tyOps.tyBtnAccDat.bRtCompl		:= FALSE;
		tyP0207OpsMagConv2.tyOps.tyBtnAccDat.bRtCompl		:= FALSE;

		tyP0003MMenu.tyMMenuBtn.tyBtnAccDat.bRtCompl		:= FALSE;
		bProdAccData	:= TRUE;
	END_IF

	//Button Appearance
	IF (p_bLFFollowerProdAccDataMnl = TRUE) OR (p_bLCSLFAccDataMnl = TRUE) OR (p_bUSHermesAAccDataMnl = TRUE) OR (p_bUSHermesBAccDataMnl = TRUE) THEN

		fbAccDatBlinkTm(IN := TRUE);

		IF fbAccDatBlinkTm.Q THEN
			fbAccDatBlinkTm(IN := FALSE);

			IF (tyP0200OpsGen.tyOps.tyBitmapAccDat.usiValueIdx = 1) THEN
				tyP0200OpsGen.tyOps.tyBitmapAccDat.usiValueIdx			:= 0;
				tyP0201OpsTravLifter.tyOps.tyBitmapAccDat.usiValueIdx	:= 0;
				tyP0202OpsMag1.tyOps.tyBitmapAccDat.usiValueIdx			:= 0;
				tyP0203OpsMag2.tyOps.tyBitmapAccDat.usiValueIdx			:= 0;
				tyP0204OpsMag3.tyOps.tyBitmapAccDat.usiValueIdx			:= 0;
				tyP0206OpsMagConv1.tyOps.tyBitmapAccDat.usiValueIdx			:= 0;
				tyP0207OpsMagConv2.tyOps.tyBitmapAccDat.usiValueIdx			:= 0;

				tyP0003MMenu.tyMMenuBtn.tyBtnAccDat.usiBitmapIdx   := 0;
			ELSE
				tyP0200OpsGen.tyOps.tyBitmapAccDat.usiValueIdx			:= 1;
				tyP0201OpsTravLifter.tyOps.tyBitmapAccDat.usiValueIdx	:= 1;
				tyP0202OpsMag1.tyOps.tyBitmapAccDat.usiValueIdx			:= 1;
				tyP0203OpsMag2.tyOps.tyBitmapAccDat.usiValueIdx			:= 1;
				tyP0204OpsMag3.tyOps.tyBitmapAccDat.usiValueIdx			:= 1;
				tyP0206OpsMagConv1.tyOps.tyBitmapAccDat.usiValueIdx			:= 1;
				tyP0207OpsMagConv2.tyOps.tyBitmapAccDat.usiValueIdx			:= 1;

				tyP0003MMenu.tyMMenuBtn.tyBtnAccDat.usiBitmapIdx   := 1;
			END_IF
		END_IF

		fUIInRtStatOff(ADR(tyP0200OpsGen.tyOps.tyBtnAccDat.uiRtStat));
		fUIInRtStatOff(ADR(tyP0201OpsTravLifter.tyOps.tyBtnAccDat.uiRtStat));
		fUIInRtStatOff(ADR(tyP0202OpsMag1.tyOps.tyBtnAccDat.uiRtStat));
		fUIInRtStatOff(ADR(tyP0203OpsMag2.tyOps.tyBtnAccDat.uiRtStat));
		fUIInRtStatOff(ADR(tyP0204OpsMag3.tyOps.tyBtnAccDat.uiRtStat));
		fUIInRtStatOff(ADR(tyP0206OpsMagConv1.tyOps.tyBtnAccDat.uiRtStat));
		fUIInRtStatOff(ADR(tyP0207OpsMagConv2.tyOps.tyBtnAccDat.uiRtStat));

		fUIInRtStatOff(ADR(tyP0200OpsGen.tyOps.tyBitmapAccDat.uiRtStat));
		fUIInRtStatOff(ADR(tyP0201OpsTravLifter.tyOps.tyBitmapAccDat.uiRtStat));
		fUIInRtStatOff(ADR(tyP0202OpsMag1.tyOps.tyBitmapAccDat.uiRtStat));
		fUIInRtStatOff(ADR(tyP0203OpsMag2.tyOps.tyBitmapAccDat.uiRtStat));
		fUIInRtStatOff(ADR(tyP0204OpsMag3.tyOps.tyBitmapAccDat.uiRtStat));
		fUIInRtStatOff(ADR(tyP0206OpsMagConv1.tyOps.tyBitmapAccDat.uiRtStat));
		fUIInRtStatOff(ADR(tyP0207OpsMagConv2.tyOps.tyBitmapAccDat.uiRtStat));

		fUIInRtStatOff(ADR(tyP0003MMenu.tyMMenuBtn.tyBtnAccDat.uiRtStat));

	ELSE

		fbAccDatBlinkTm(IN := FALSE);

		tyP0200OpsGen.tyOps.tyBitmapAccDat.usiValueIdx			:= 0;
		tyP0201OpsTravLifter.tyOps.tyBitmapAccDat.usiValueIdx	:= 0;
		tyP0202OpsMag1.tyOps.tyBitmapAccDat.usiValueIdx			:= 0;
		tyP0203OpsMag2.tyOps.tyBitmapAccDat.usiValueIdx			:= 0;
		tyP0204OpsMag3.tyOps.tyBitmapAccDat.usiValueIdx			:= 0;
		tyP0206OpsMagConv1.tyOps.tyBitmapAccDat.usiValueIdx			:= 0;
		tyP0207OpsMagConv2.tyOps.tyBitmapAccDat.usiValueIdx			:= 0;

		tyP0003MMenu.tyMMenuBtn.tyBtnAccDat.usiBitmapIdx := 0;

		fUIInRtStatHide(ADR(tyP0200OpsGen.tyOps.tyBtnAccDat.uiRtStat));
		fUIInRtStatHide(ADR(tyP0201OpsTravLifter.tyOps.tyBtnAccDat.uiRtStat));
		fUIInRtStatHide(ADR(tyP0202OpsMag1.tyOps.tyBtnAccDat.uiRtStat));
		fUIInRtStatHide(ADR(tyP0203OpsMag2.tyOps.tyBtnAccDat.uiRtStat));
		fUIInRtStatHide(ADR(tyP0204OpsMag3.tyOps.tyBtnAccDat.uiRtStat));
		fUIInRtStatHide(ADR(tyP0206OpsMagConv1.tyOps.tyBtnAccDat.uiRtStat));
		fUIInRtStatHide(ADR(tyP0207OpsMagConv2.tyOps.tyBtnAccDat.uiRtStat));

		fUIInRtStatHide(ADR(tyP0200OpsGen.tyOps.tyBitmapAccDat.uiRtStat));
		fUIInRtStatHide(ADR(tyP0201OpsTravLifter.tyOps.tyBitmapAccDat.uiRtStat));
		fUIInRtStatHide(ADR(tyP0202OpsMag1.tyOps.tyBitmapAccDat.uiRtStat));
		fUIInRtStatHide(ADR(tyP0203OpsMag2.tyOps.tyBitmapAccDat.uiRtStat));
		fUIInRtStatHide(ADR(tyP0204OpsMag3.tyOps.tyBitmapAccDat.uiRtStat));
		fUIInRtStatHide(ADR(tyP0206OpsMagConv1.tyOps.tyBitmapAccDat.uiRtStat));
		fUIInRtStatHide(ADR(tyP0207OpsMagConv2.tyOps.tyBitmapAccDat.uiRtStat));

		fUIInRtStatHide(ADR(tyP0003MMenu.tyMMenuBtn.tyBtnAccDat.uiRtStat));
	END_IF

END_ACTION
```
